KUKA KRL program: EPS_2_251455_MH14A_A_20251003045101.src

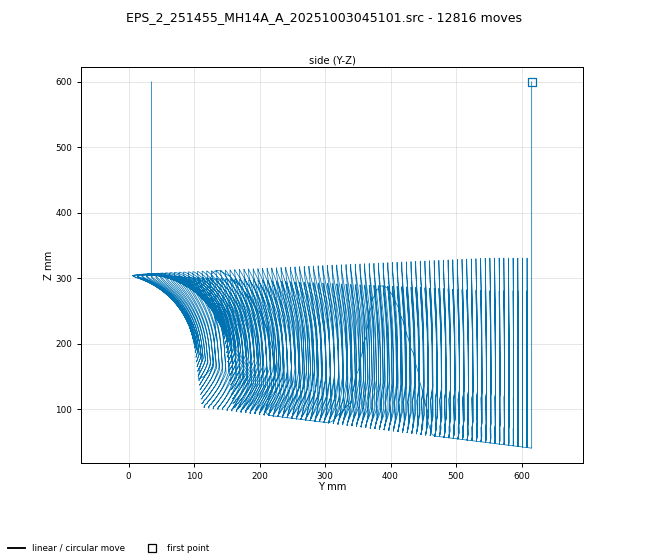
[picture p0: tool path of EPS_2_251455_MH14A_A_20251003045101.src, 12816 of 12818 moves have a stored position in this frame; points joined in program order, loops and branches not executed]
&ACCESS RVP
&REL 4
&COMMENT QRS 19112012
&PARAM EDITMASK = *
DEF PART()
EXT BAS (BAS_COMMAND :IN,REAL :IN )
INT I
BAS (#INITMOV,0 )

;KUKA QRS Post kuka4.cps  Date:22-06-2017 !

File_ID=2870

QRS_PRE_INIT()

;Init var - Until changes are made in qrs_pre_init
Outlet_Square_prg=0
Inlet_1_Square_prg=0
Inlet_2_Square_prg=0
Inlet_3_Square_prg=0
Inlet_4_Square_prg=0
Inlet_5_Square_prg=0

Outlet_1={X 0.000, Y 551.740, Z 230.500, B 0.000, E1 0.000 }
Inlet_1={X 0.000, Y 555.300, Z 180.500, B 0.000, E1 187.000 }
Outlet_1_type=201
Inlet_1_type=201
;QRS#1=Sidecore dimensions
;QRS#2=200-8" PVC SDR 35
;QRS#3=200-8" PVC SDR 35
;QRS#4=
;QRS#5=
;QRS#6=
;QRS#7=
;QRS#8=
;QRS#9=12-08 PSX
;QRS#10=12-08 PSX
;QRS#11=
;QRS#12=
;QRS#13=
;QRS#14=
;QRS#15=
;QRS#16=1220x127x610 2'
;QRS#17=EPS Height
;QRS#18=331
;QRS#19=*
;QRS#20= UPDATED VERSION 22-06-2017
;QRS#21=*
Outlet_Square=0100
Inlet_1_Square=0100
Inlet_2_Square=0
Inlet_3_Square=0
Inlet_4_Square=0
Inlet_5_Square=0
Mill_Square=1
Outlet_Square_Prg=204
Inlet_1_Square_prg=204

QRS_INIT()

$ADVANCE=5

; T1
PTP {E1 173.635,E2 173.635}
PTP {X 0,Y 615.458,A -85,B 0,C 180,E1 173.635,E2 173.635,E3 0,E4 0,E5 0,E6 0}
QRS_SPEED_INIT()
LIN {X 0,Y 615.458,Z 600,A -85,B 0,C 180,E1 173.635,E2 173.635,E3 0,E4 0,E5 0,E6 0} C_VEL
LIN {X 0,Y 615.458,Z 50.874,A -85,B 0,C 180,E1 173.635,E2 173.635} C_VEL
LIN {X 0,Y 615.458,Z 42.693,A -85,B 0,C 180,E1 173.635,E2 173.635} C_VEL
LIN {X 0,Y 615.454,Z 40.693,A -85,B 0,C 180,E1 173.449,E2 173.449} C_VEL
LIN {X 0,Y 615.495,Z 40.685,A -85,B 0,C 180,E1 170.801,E2 170.801} C_VEL
LIN {X 0,Y 615.481,Z 40.699,A -85,B 0,C 180,E1 168.139,E2 168.139} C_VEL
LIN {X 0,Y 615.455,Z 40.691,A -85,B 0,C 180,E1 165.45,E2 165.45} C_VEL
LIN {X 0,Y 615.493,Z 40.692,A -85,B 0,C 180,E1 162.729,E2 162.729} C_VEL
LIN {X 0,Y 615.454,Z 40.694,A -85,B 0,C 180,E1 159.966,E2 159.966} C_VEL
LIN {X 0,Y 615.455,Z 40.69,A -85,B 0,C 180,E1 157.661,E2 157.661} C_VEL
LIN {X 0,Y 615.495,Z 40.691,A -85,B 0,C 180,E1 155.008,E2 155.008} C_VEL
LIN {X 0,Y 615.45,Z 40.693,A -85,B 0,C 180,E1 152.083,E2 152.083} C_VEL
LIN {X 0,Y 615.452,Z 40.691,A -85,B 0,C 180,E1 149.838,E2 149.838} C_VEL
LIN {X 0,Y 615.478,Z 40.688,A -85,B 0,C 180,E1 147.542,E2 147.542} C_VEL
LIN {X 0,Y 615.495,Z 40.695,A -85,B 0,C 180,E1 145.185,E2 145.185} C_VEL
LIN {X 0,Y 615.465,Z 40.697,A -85,B 0,C 180,E1 142.756,E2 142.756} C_VEL
LIN {X 0,Y 615.448,Z 40.692,A -85,B 0,C 180,E1 140.246,E2 140.246} C_VEL
LIN {X 0,Y 615.499,Z 40.688,A -85,B 0,C 180,E1 137.647,E2 137.647} C_VEL
LIN {X 0,Y 615.458,Z 40.697,A -85,B 0,C 180,E1 134.928,E2 134.928} C_VEL
LIN {X 0,Y 615.451,Z 40.691,A -85,B 0,C 180,E1 132.356,E2 132.356} C_VEL
LIN {X 0,Y 615.495,Z 40.693,A -85,B 0,C 180,E1 129.749,E2 129.749} C_VEL
LIN {X 0,Y 615.445,Z 40.695,A -85,B 0,C 180,E1 126.931,E2 126.931} C_VEL
LIN {X 0,Y 615.444,Z 40.693,A -85,B 0,C 180,E1 124.694,E2 124.694} C_VEL
LIN {X 0,Y 615.472,Z 40.69,A -85,B 0,C 180,E1 122.328,E2 122.328} C_VEL
LIN {X 0,Y 615.455,Z 40.697,A -85,B 0,C 180,E1 119.408,E2 119.408} C_VEL
LIN {X 0,Y 615.439,Z 40.695,A -85,B 0,C 180,E1 117.035,E2 117.035} C_VEL
LIN {X 0,Y 615.491,Z 40.692,A -85,B 0,C 180,E1 114.272,E2 114.272} C_VEL
LIN {X 0,Y 615.497,Z 40.698,A -85,B 0,C 180,E1 112.136,E2 112.136} C_VEL
LIN {X 0,Y 615.487,Z 40.7,A -85,B 0,C 180,E1 110.033,E2 110.033} C_VEL
LIN {X 0,Y 615.47,Z 40.699,A -85,B 0,C 180,E1 107.957,E2 107.957} C_VEL
LIN {X 0,Y 615.457,Z 40.699,A -85,B 0,C 180,E1 105.906,E2 105.906} C_VEL
LIN {X 0,Y 615.451,Z 40.698,A -85,B 0,C 180,E1 103.875,E2 103.875} C_VEL
LIN {X 0,Y 615.446,Z 40.697,A -85,B 0,C 180,E1 101.861,E2 101.861} C_VEL
LIN {X 0,Y 615.467,Z 40.868,A -85,B 0,C 180,E1 100.958,E2 100.958} C_VEL
LIN {X 0,Y 615.443,Z 56.59,A -85,B 0,C 180,E1 98.206,E2 98.206} C_VEL
LIN {X 0,Y 615.459,Z 70.383,A -85,B 0,C 180,E1 95.816,E2 95.816} C_VEL
LIN {X 0,Y 615.474,Z 176.897,A -85,B 0,C 180,E1 94.543,E2 94.543} C_VEL
LIN {X 0,Y 615.468,Z 189.97,A -85,B 0,C 180,E1 94.256,E2 94.256} C_VEL
LIN {X 0,Y 615.485,Z 202.502,A -85,B 0,C 180,E1 93.846,E2 93.846} C_VEL
LIN {X 0,Y 615.485,Z 213.691,A -85,B 0,C 180,E1 93.355,E2 93.355} C_VEL
LIN {X 0,Y 615.491,Z 225.253,A -85,B 0,C 180,E1 92.7,E2 92.7} C_VEL
LIN {X 0,Y 615.498,Z 236.649,A -85,B 0,C 180,E1 91.881,E2 91.881} C_VEL
LIN {X 0,Y 615.498,Z 244.983,A -85,B 0,C 180,E1 91.145,E2 91.145} C_VEL
LIN {X 0,Y 615.498,Z 254.024,A -85,B 0,C 180,E1 90.163,E2 90.163} C_VEL
LIN {X 0,Y 615.498,Z 261.318,A -85,B 0,C 180,E1 89.182,E2 89.182} C_VEL
LIN {X 0,Y 615.497,Z 268.049,A -85,B 0,C 180,E1 88.037,E2 88.037} C_VEL
LIN {X 0,Y 615.496,Z 272.502,A -85,B 0,C 180,E1 87.054,E2 87.054} C_VEL
LIN {X 0,Y 615.496,Z 275.893,A -85,B 0,C 180,E1 86.071,E2 86.071} C_VEL
LIN {X 0,Y 615.498,Z 277.586,A -85,B 0,C 180,E1 85.415,E2 85.415} C_VEL
LIN {X 0,Y 615.497,Z 279.772,A -85,B 0,C 180,E1 84.101,E2 84.101} C_VEL
LIN {X 0,Y 615.495,Z 280.285,A -85,B 0,C 180,E1 83.42,E2 83.42} C_VEL
LIN {X 0,Y 615.494,Z 280.049,A -85,B 0,C 180,E1 82.124,E2 82.124} C_VEL
LIN {X 0,Y 615.496,Z 279.365,A -85,B 0,C 180,E1 81.463,E2 81.463} C_VEL
LIN {X 0,Y 615.496,Z 278.251,A -85,B 0,C 180,E1 80.801,E2 80.801} C_VEL
LIN {X 0,Y 615.496,Z 276.7,A -85,B 0,C 180,E1 80.138,E2 80.138} C_VEL
LIN {X 0,Y 615.496,Z 273.454,A -85,B 0,C 180,E1 79.11,E2 79.11} C_VEL
LIN {X 0,Y 615.496,Z 269.345,A -85,B 0,C 180,E1 78.139,E2 78.139} C_VEL
LIN {X 0,Y 615.496,Z 262.875,A -85,B 0,C 180,E1 76.967,E2 76.967} C_VEL
LIN {X 0,Y 615.497,Z 255.382,A -85,B 0,C 180,E1 75.912,E2 75.912} C_VEL
LIN {X 0,Y 615.498,Z 246.759,A -85,B 0,C 180,E1 74.943,E2 74.943} C_VEL
LIN {X 0,Y 615.497,Z 237.478,A -85,B 0,C 180,E1 74.095,E2 74.095} C_VEL
LIN {X 0,Y 615.487,Z 227.053,A -85,B 0,C 180,E1 73.328,E2 73.328} C_VEL
LIN {X 0,Y 615.468,Z 215.403,A -85,B 0,C 180,E1 72.643,E2 72.643} C_VEL
LIN {X 0,Y 615.492,Z 203.097,A -85,B 0,C 180,E1 72.086,E2 72.086} C_VEL
LIN {X 0,Y 615.489,Z 190.885,A -85,B 0,C 180,E1 71.679,E2 71.679} C_VEL
LIN {X 0,Y 615.489,Z 177.332,A -85,B 0,C 180,E1 71.375,E2 71.375} C_VEL
LIN {X 0,Y 615.475,Z 70.399,A -85,B 0,C 180,E1 70.097,E2 70.097} C_VEL
LIN {X 0,Y 615.495,Z 54.86,A -85,B 0,C 180,E1 67.405,E2 67.405} C_VEL
LIN {X 0,Y 615.436,Z 40.698,A -85,B 0,C 180,E1 64.901,E2 64.901} C_VEL
LIN {X 0,Y 615.428,Z 40.698,A -85,B 0,C 180,E1 62.82,E2 62.82} C_VEL
LIN {X 0,Y 615.428,Z 40.697,A -85,B 0,C 180,E1 60.59,E2 60.59} C_VEL
LIN {X 0,Y 615.446,Z 40.696,A -85,B 0,C 180,E1 58.312,E2 58.312} C_VEL
LIN {X 0,Y 615.494,Z 40.696,A -85,B 0,C 180,E1 55.978,E2 55.978} C_VEL
LIN {X 0,Y 615.454,Z 40.699,A -85,B 0,C 180,E1 53.573,E2 53.573} C_VEL
LIN {X 0,Y 615.42,Z 40.699,A -85,B 0,C 180,E1 50.946,E2 50.946} C_VEL
LIN {X 0,Y 615.449,Z 40.698,A -85,B 0,C 180,E1 48.523,E2 48.523} C_VEL
LIN {X 0,Y 615.452,Z 40.7,A -85,B 0,C 180,E1 45.847,E2 45.847} C_VEL
LIN {X 0,Y 615.461,Z 40.7,A -85,B 0,C 180,E1 43.995,E2 43.995} C_VEL
LIN {X 0,Y 615.415,Z 40.7,A -85,B 0,C 180,E1 41.48,E2 41.48} C_VEL
LIN {X 0,Y 615.438,Z 40.7,A -85,B 0,C 180,E1 38.909,E2 38.909} C_VEL
LIN {X 0,Y 615.469,Z 40.704,A -85,B 0,C 180,E1 36.426,E2 36.426} C_VEL
LIN {X 0,Y 615.435,Z 40.699,A -85,B 0,C 180,E1 34.026,E2 34.026} C_VEL
LIN {X 0,Y 615.419,Z 40.699,A -85,B 0,C 180,E1 31.69,E2 31.69} C_VEL
LIN {X 0,Y 615.426,Z 40.7,A -85,B 0,C 180,E1 29.41,E2 29.41} C_VEL
LIN {X 0,Y 615.473,Z 40.7,A -85,B 0,C 180,E1 27.042,E2 27.042} C_VEL
LIN {X 0,Y 615.437,Z 40.697,A -85,B 0,C 180,E1 24.274,E2 24.274} C_VEL
LIN {X 0,Y 615.428,Z 40.697,A -85,B 0,C 180,E1 22.139,E2 22.139} C_VEL
LIN {X 0,Y 615.426,Z 40.697,A -85,B 0,C 180,E1 20.035,E2 20.035} C_VEL
LIN {X 0,Y 615.486,Z 40.701,A -85,B 0,C 180,E1 17.271,E2 17.271} C_VEL
LIN {X 0,Y 615.439,Z 40.695,A -85,B 0,C 180,E1 14.55,E2 14.55} C_VEL
LIN {X 0,Y 615.437,Z 40.695,A -85,B 0,C 180,E1 12.531,E2 12.531} C_VEL
LIN {X 0,Y 615.436,Z 40.695,A -85,B 0,C 180,E1 10.528,E2 10.528} C_VEL
LIN {X 0,Y 615.435,Z 40.695,A -85,B 0,C 180,E1 8.538,E2 8.538} C_VEL
LIN {X 0,Y 615.459,Z 40.7,A -85,B 0,C 180,E1 5.899,E2 5.899} C_VEL
LIN {X 0,Y 615.478,Z 40.692,A -85,B 0,C 180,E1 3.273,E2 3.273} C_VEL
LIN {X 0,Y 615.438,Z 40.695,A -85,B 0,C 180,E1 0.654,E2 0.654} C_VEL
LIN {X 0,Y 615.481,Z 40.699,A -85,B 0,C 180,E1 -1.963,E2 -1.963} C_VEL
LIN {X 0,Y 615.473,Z 40.69,A -85,B 0,C 180,E1 -4.585,E2 -4.585} C_VEL
LIN {X 0,Y 615.443,Z 40.695,A -85,B 0,C 180,E1 -7.216,E2 -7.216} C_VEL
LIN {X 0,Y 615.499,Z 40.699,A -85,B 0,C 180,E1 -9.862,E2 -9.862} C_VEL
LIN {X 0,Y 615.46,Z 40.69,A -85,B 0,C 180,E1 -12.531,E2 -12.531} C_VEL
LIN {X 0,Y 615.456,Z 40.691,A -85,B 0,C 180,E1 -14.55,E2 -14.55} C_VEL
LIN {X 0,Y 615.45,Z 40.692,A -85,B 0,C 180,E1 -16.588,E2 -16.588} C_VEL
LIN {X 0,Y 615.448,Z 40.693,A -85,B 0,C 180,E1 -18.647,E2 -18.647} C_VEL
LIN {X 0,Y 615.497,Z 40.7,A -85,B 0,C 180,E1 -21.432,E2 -21.432} C_VEL
LIN {X 0,Y 615.459,Z 40.69,A -85,B 0,C 180,E1 -24.273,E2 -24.273} C_VEL
LIN {X 0,Y 615.453,Z 40.692,A -85,B 0,C 180,E1 -26.446,E2 -26.446} C_VEL
LIN {X 0,Y 615.458,Z 40.695,A -85,B 0,C 180,E1 -28.66,E2 -28.66} C_VEL
LIN {X 0,Y 615.486,Z 40.703,A -85,B 0,C 180,E1 -31.085,E2 -31.085} C_VEL
LIN {X 0,Y 615.461,Z 40.689,A -85,B 0,C 180,E1 -34.024,E2 -34.024} C_VEL
LIN {X 0,Y 615.463,Z 40.695,A -85,B 0,C 180,E1 -36.427,E2 -36.427} C_VEL
LIN {X 0,Y 615.492,Z 40.693,A -85,B 0,C 180,E1 -39.062,E2 -39.062} C_VEL
LIN {X 0,Y 615.487,Z 40.684,A -85,B 0,C 180,E1 -41.474,E2 -41.474} C_VEL
LIN {X 0,Y 615.463,Z 40.695,A -85,B 0,C 180,E1 -44.152,E2 -44.152} C_VEL
LIN {X 0,Y 615.489,Z 40.689,A -85,B 0,C 180,E1 -46.953,E2 -46.953} C_VEL
LIN {X 0,Y 615.474,Z 40.686,A -85,B 0,C 180,E1 -49.392,E2 -49.392} C_VEL
LIN {X 0,Y 615.469,Z 40.696,A -85,B 0,C 180,E1 -51.99,E2 -51.99} C_VEL
LIN {X 0,Y 615.493,Z 40.697,A -85,B 0,C 180,E1 -54.384,E2 -54.384} C_VEL
LIN {X 0,Y 615.486,Z 40.687,A -85,B 0,C 180,E1 -56.763,E2 -56.763} C_VEL
LIN {X 0,Y 615.478,Z 40.685,A -85,B 0,C 180,E1 -59.079,E2 -59.079} C_VEL
LIN {X 0,Y 615.471,Z 40.693,A -85,B 0,C 180,E1 -61.553,E2 -61.553} C_VEL
LIN {X 0,Y 615.487,Z 40.687,A -85,B 0,C 180,E1 -64.432,E2 -64.432} C_VEL
LIN {X 0,Y 615.47,Z 40.821,A -85,B 0,C 180,E1 -67.066,E2 -67.066} C_VEL
LIN {X 0,Y 615.461,Z 60.773,A -85,B 0,C 180,E1 -69.706,E2 -69.706} C_VEL
LIN {X 0,Y 615.488,Z 82.668,A -85,B 0,C 180,E1 -72.558,E2 -72.558} C_VEL
LIN {X 0,Y 615.467,Z 103.89,A -85,B 0,C 180,E1 -75.281,E2 -75.281} C_VEL
LIN {X 0,Y 615.452,Z 118.299,A -85,B 0,C 180,E1 -77.113,E2 -77.113} C_VEL
LIN {X 0,Y 615.492,Z 226.816,A -85,B 0,C 180,E1 -78.411,E2 -78.411} C_VEL
LIN {X 0,Y 615.48,Z 239.337,A -85,B 0,C 180,E1 -78.681,E2 -78.681} C_VEL
LIN {X 0,Y 615.489,Z 252.607,A -85,B 0,C 180,E1 -79.113,E2 -79.113} C_VEL
LIN {X 0,Y 615.475,Z 264.475,A -85,B 0,C 180,E1 -79.639,E2 -79.639} C_VEL
LIN {X 0,Y 615.492,Z 275.991,A -85,B 0,C 180,E1 -80.304,E2 -80.304} C_VEL
LIN {X 0,Y 615.499,Z 286.338,A -85,B 0,C 180,E1 -81.05,E2 -81.05} C_VEL
LIN {X 0,Y 615.497,Z 294.809,A -85,B 0,C 180,E1 -81.794,E2 -81.794} C_VEL
LIN {X 0,Y 615.498,Z 302.604,A -85,B 0,C 180,E1 -82.619,E2 -82.619} C_VEL
LIN {X 0,Y 615.496,Z 310.201,A -85,B 0,C 180,E1 -83.608,E2 -83.608} C_VEL
LIN {X 0,Y 615.498,Z 317.203,A -85,B 0,C 180,E1 -84.759,E2 -84.759} C_VEL
LIN {X 0,Y 615.493,Z 321.85,A -85,B 0,C 180,E1 -85.743,E2 -85.743} C_VEL
LIN {X 0,Y 615.494,Z 325.398,A -85,B 0,C 180,E1 -86.727,E2 -86.727} C_VEL
LIN {X 0,Y 615.497,Z 327.232,A -85,B 0,C 180,E1 -87.382,E2 -87.382} C_VEL
LIN {X 0,Y 615.5,Z 328.607,A -85,B 0,C 180,E1 -88.037,E2 -88.037} C_VEL
LIN {X 0,Y 615.496,Z 330.173,A -85,B 0,C 180,E1 -89.346,E2 -89.346} C_VEL
LIN {X 0,Y 615.494,Z 330.389,A -85,B 0,C 180,E1 -90,E2 -90} C_VEL
LIN {X 0,Y 615.495,Z 329.58,A -85,B 0,C 180,E1 -91.308,E2 -91.308} C_VEL
LIN {X 0,Y 615.5,Z 328.608,A -85,B 0,C 180,E1 -91.963,E2 -91.963} C_VEL
LIN {X 0,Y 615.497,Z 327.233,A -85,B 0,C 180,E1 -92.618,E2 -92.618} C_VEL
LIN {X 0,Y 615.496,Z 324.35,A -85,B 0,C 180,E1 -93.6,E2 -93.6} C_VEL
LIN {X 0,Y 615.498,Z 320.442,A -85,B 0,C 180,E1 -94.584,E2 -94.584} C_VEL
LIN {X 0,Y 615.499,Z 315.406,A -85,B 0,C 180,E1 -95.569,E2 -95.569} C_VEL
LIN {X 0,Y 615.497,Z 308.869,A -85,B 0,C 180,E1 -96.583,E2 -96.583} C_VEL
LIN {X 0,Y 615.497,Z 301.135,A -85,B 0,C 180,E1 -97.545,E2 -97.545} C_VEL
LIN {X 0,Y 615.498,Z 293.047,A -85,B 0,C 180,E1 -98.371,E2 -98.371} C_VEL
LIN {X 0,Y 615.499,Z 283.17,A -85,B 0,C 180,E1 -99.198,E2 -99.198} C_VEL
LIN {X 0,Y 615.484,Z 271.985,A -85,B 0,C 180,E1 -99.945,E2 -99.945} C_VEL
LIN {X 0,Y 615.481,Z 261.027,A -85,B 0,C 180,E1 -100.527,E2 -100.527} C_VEL
LIN {X 0,Y 615.481,Z 248.487,A -85,B 0,C 180,E1 -101.04,E2 -101.04} C_VEL
LIN {X 0,Y 615.482,Z 236.074,A -85,B 0,C 180,E1 -101.401,E2 -101.401} C_VEL
LIN {X 0,Y 615.497,Z 222.476,A -85,B 0,C 180,E1 -101.652,E2 -101.652} C_VEL
LIN {X 0,Y 615.452,Z 118.302,A -85,B 0,C 180,E1 -102.887,E2 -102.887} C_VEL
LIN {X 0,Y 615.488,Z 95.935,A -85,B 0,C 180,E1 -105.735,E2 -105.735} C_VEL
LIN {X 0,Y 615.456,Z 75.012,A -85,B 0,C 180,E1 -108.435,E2 -108.435} C_VEL
LIN {X 0,Y 615.489,Z 54.783,A -85,B 0,C 180,E1 -111.081,E2 -111.081} C_VEL
LIN {X 0,Y 615.472,Z 40.688,A -85,B 0,C 180,E1 -112.978,E2 -112.978} C_VEL
LIN {X 0,Y 615.485,Z 40.691,A -85,B 0,C 180,E1 -115.716,E2 -115.716} C_VEL
LIN {X 0,Y 615.473,Z 40.693,A -85,B 0,C 180,E1 -118.447,E2 -118.447} C_VEL
LIN {X 0,Y 615.485,Z 40.684,A -85,B 0,C 180,E1 -121.085,E2 -121.085} C_VEL
LIN {X 0,Y 615.483,Z 40.698,A -85,B 0,C 180,E1 -124.022,E2 -124.022} C_VEL
LIN {X 0,Y 615.468,Z 40.69,A -85,B 0,C 180,E1 -126.426,E2 -126.426} C_VEL
LIN {X 0,Y 615.492,Z 40.685,A -85,B 0,C 180,E1 -129.062,E2 -129.062} C_VEL
LIN {X 0,Y 615.49,Z 40.697,A -85,B 0,C 180,E1 -131.473,E2 -131.473} C_VEL
LIN {X 0,Y 615.467,Z 40.691,A -85,B 0,C 180,E1 -134.151,E2 -134.151} C_VEL
LIN {X 0,Y 615.487,Z 40.688,A -85,B 0,C 180,E1 -136.952,E2 -136.952} C_VEL
LIN {X 0,Y 615.486,Z 40.702,A -85,B 0,C 180,E1 -139.393,E2 -139.393} C_VEL
LIN {X 0,Y 615.465,Z 40.69,A -85,B 0,C 180,E1 -141.991,E2 -141.991} C_VEL
LIN {X 0,Y 615.489,Z 40.683,A -85,B 0,C 180,E1 -144.384,E2 -144.384} C_VEL
LIN {X 0,Y 615.489,Z 40.691,A -85,B 0,C 180,E1 -146.764,E2 -146.764} C_VEL
LIN {X 0,Y 615.49,Z 40.702,A -85,B 0,C 180,E1 -149.08,E2 -149.08} C_VEL
LIN {X 0,Y 615.464,Z 40.692,A -85,B 0,C 180,E1 -151.554,E2 -151.554} C_VEL
LIN {X 0,Y 615.496,Z 40.684,A -85,B 0,C 180,E1 -154.285,E2 -154.285} C_VEL
LIN {X 0,Y 615.471,Z 40.696,A -85,B 0,C 180,E1 -157.155,E2 -157.155} C_VEL
LIN {X 0,Y 615.483,Z 40.685,A -85,B 0,C 180,E1 -159.967,E2 -159.967} C_VEL
LIN {X 0,Y 615.49,Z 40.699,A -85,B 0,C 180,E1 -162.73,E2 -162.73} C_VEL
LIN {X 0,Y 615.464,Z 40.689,A -85,B 0,C 180,E1 -165.45,E2 -165.45} C_VEL
LIN {X 0,Y 615.491,Z 40.691,A -85,B 0,C 180,E1 -168.139,E2 -168.139} C_VEL
LIN {X 0,Y 615.465,Z 40.695,A -85,B 0,C 180,E1 -170.801,E2 -170.801} C_VEL
LIN {X 0,Y 615.476,Z 40.686,A -85,B 0,C 180,E1 -173.443,E2 -173.443} C_VEL
LIN {X 0,Y 615.492,Z 40.697,A -85,B 0,C 180,E1 -176.072,E2 -176.072} C_VEL
LIN {X 0,Y 615.457,Z 40.694,A -85,B 0,C 180,E1 -178.691,E2 -178.691} C_VEL
LIN {X 0,Y 615.483,Z 40.685,A -85,B 0,C 180,E1 -181.309,E2 -181.309} C_VEL
LIN {X 0,Y 615.488,Z 40.701,A -85,B 0,C 180,E1 -183.929,E2 -183.929} C_VEL
LIN {X 0,Y 615.454,Z 40.693,A -85,B 0,C 180,E1 -186.551,E2 -186.551} C_VEL
LIN {X 0,Y 614.802,Z 40.835,A -85,B 0,C 180,E1 -187.097,E2 -187.097} C_VEL
LIN {X 0,Y 611.99,Z 41.255,A -85,B 0,C 180,E1 -187.984,E2 -187.984} C_VEL
LIN {X 0,Y 609.6,Z 41.562,A -85,B 0,C 180,E1 -188.696,E2 -188.696} C_VEL
LIN {X 0,Y 608.559,Z 41.678,A -85,B 0,C 180,E1 -189.246,E2 -189.246} C_VEL
LIN {X 0,Y 608.467,Z 41.689,A -85,B 0,C 180,E1 -189.432,E2 -189.432} C_VEL
LIN {X 0,Y 608.452,Z 41.693,A -85,B 0,C 180,E1 -192,E2 -192} C_VEL
LIN {X 0,Y 608.429,Z 41.691,A -85,B 0,C 180,E1 -194.722,E2 -194.722} C_VEL
LIN {X 0,Y 608.45,Z 41.697,A -85,B 0,C 180,E1 -197.477,E2 -197.477} C_VEL
LIN {X 0,Y 608.437,Z 41.69,A -85,B 0,C 180,E1 -200.275,E2 -200.275} C_VEL
LIN {X 0,Y 608.429,Z 41.691,A -85,B 0,C 180,E1 -202.47,E2 -202.47} C_VEL
LIN {X 0,Y 608.446,Z 41.699,A -85,B 0,C 180,E1 -205.302,E2 -205.302} C_VEL
LIN {X 0,Y 608.437,Z 41.695,A -85,B 0,C 180,E1 -207.519,E2 -207.519} C_VEL
LIN {X 0,Y 608.418,Z 41.692,A -85,B 0,C 180,E1 -209.964,E2 -209.964} C_VEL
LIN {X 0,Y 608.455,Z 41.69,A -85,B 0,C 180,E1 -212.522,E2 -212.522} C_VEL
LIN {X 0,Y 608.427,Z 41.696,A -85,B 0,C 180,E1 -215.279,E2 -215.279} C_VEL
LIN {X 0,Y 608.446,Z 41.689,A -85,B 0,C 180,E1 -217.748,E2 -217.748} C_VEL
LIN {X 0,Y 608.443,Z 41.692,A -85,B 0,C 180,E1 -220.328,E2 -220.328} C_VEL
LIN {X 0,Y 608.437,Z 41.696,A -85,B 0,C 180,E1 -222.962,E2 -222.962} C_VEL
LIN {X 0,Y 608.431,Z 41.69,A -85,B 0,C 180,E1 -225.739,E2 -225.739} C_VEL
LIN {X 0,Y 608.451,Z 41.689,A -85,B 0,C 180,E1 -227.938,E2 -227.938} C_VEL
LIN {X 0,Y 608.43,Z 41.697,A -85,B 0,C 180,E1 -230.708,E2 -230.708} C_VEL
LIN {X 0,Y 608.416,Z 41.693,A -85,B 0,C 180,E1 -233.082,E2 -233.082} C_VEL
LIN {X 0,Y 608.446,Z 41.689,A -85,B 0,C 180,E1 -235.529,E2 -235.529} C_VEL
LIN {X 0,Y 608.458,Z 41.691,A -85,B 0,C 180,E1 -237.905,E2 -237.905} C_VEL
LIN {X 0,Y 608.482,Z 41.694,A -85,B 0,C 180,E1 -240.221,E2 -240.221} C_VEL
LIN {X 0,Y 608.421,Z 41.693,A -85,B 0,C 180,E1 -242.804,E2 -242.804} C_VEL
LIN {X 0,Y 608.44,Z 41.691,A -85,B 0,C 180,E1 -245.429,E2 -245.429} C_VEL
LIN {X 0,Y 608.448,Z 41.692,A -85,B 0,C 180,E1 -248.308,E2 -248.308} C_VEL
LIN {X 0,Y 608.425,Z 41.693,A -85,B 0,C 180,E1 -250.429,E2 -250.429} C_VEL
LIN {X 0,Y 608.436,Z 41.692,A -85,B 0,C 180,E1 -253.216,E2 -253.216} C_VEL
LIN {X 0,Y 608.435,Z 41.695,A -85,B 0,C 180,E1 -255.998,E2 -255.998} C_VEL
LIN {X 0,Y 608.437,Z 41.694,A -85,B 0,C 180,E1 -258,E2 -258} C_VEL
LIN {X 0,Y 608.468,Z 41.758,A -85,B 0,C 180,E1 -258.971,E2 -258.971} C_VEL
LIN {X 0,Y 608.433,Z 57.206,A -85,B 0,C 180,E1 -261.698,E2 -261.698} C_VEL
LIN {X 0,Y 608.433,Z 70.587,A -85,B 0,C 180,E1 -264.033,E2 -264.033} C_VEL
LIN {X 0,Y 608.55,Z 153.667,A -85,B 0,C 180,E1 -265.031,E2 -265.031} C_VEL
LIN {X 0,Y 608.52,Z 178.093,A -85,B 0,C 180,E1 -265.342,E2 -265.342} C_VEL
LIN {X 0,Y 608.528,Z 191.538,A -85,B 0,C 180,E1 -265.653,E2 -265.653} C_VEL
LIN {X 0,Y 608.513,Z 203.71,A -85,B 0,C 180,E1 -266.068,E2 -266.068} C_VEL
LIN {X 0,Y 608.493,Z 215.437,A -85,B 0,C 180,E1 -266.607,E2 -266.607} C_VEL
LIN {X 0,Y 608.495,Z 226.702,A -85,B 0,C 180,E1 -267.269,E2 -267.269} C_VEL
LIN {X 0,Y 608.472,Z 236.896,A -85,B 0,C 180,E1 -268.014,E2 -268.014} C_VEL
LIN {X 0,Y 608.479,Z 246.116,A -85,B 0,C 180,E1 -268.842,E2 -268.842} C_VEL
LIN {X 0,Y 608.469,Z 255.057,A -85,B 0,C 180,E1 -269.835,E2 -269.835} C_VEL
LIN {X 0,Y 608.448,Z 262.293,A -85,B 0,C 180,E1 -270.827,E2 -270.827} C_VEL
LIN {X 0,Y 608.443,Z 268.932,A -85,B 0,C 180,E1 -271.986,E2 -271.986} C_VEL
LIN {X 0,Y 608.451,Z 273.336,A -85,B 0,C 180,E1 -272.98,E2 -272.98} C_VEL
LIN {X 0,Y 608.433,Z 276.683,A -85,B 0,C 180,E1 -273.974,E2 -273.974} C_VEL
LIN {X 0,Y 608.431,Z 278.346,A -85,B 0,C 180,E1 -274.638,E2 -274.638} C_VEL
LIN {X 0,Y 608.433,Z 280.473,A -85,B 0,C 180,E1 -275.967,E2 -275.967} C_VEL
LIN {X 0,Y 608.43,Z 280.91,A -85,B 0,C 180,E1 -276.633,E2 -276.633} C_VEL
LIN {X 0,Y 608.419,Z 280.6,A -85,B 0,C 180,E1 -277.968,E2 -277.968} C_VEL
LIN {X 0,Y 608.422,Z 279.854,A -85,B 0,C 180,E1 -278.637,E2 -278.637} C_VEL
LIN {X 0,Y 608.421,Z 278.659,A -85,B 0,C 180,E1 -279.307,E2 -279.307} C_VEL
LIN {X 0,Y 608.433,Z 276.089,A -85,B 0,C 180,E1 -280.314,E2 -280.314} C_VEL
LIN {X 0,Y 608.43,Z 272.482,A -85,B 0,C 180,E1 -281.325,E2 -281.325} C_VEL
LIN {X 0,Y 608.459,Z 267.726,A -85,B 0,C 180,E1 -282.339,E2 -282.339} C_VEL
LIN {X 0,Y 608.459,Z 260.513,A -85,B 0,C 180,E1 -283.527,E2 -283.527} C_VEL
LIN {X 0,Y 608.459,Z 252.619,A -85,B 0,C 180,E1 -284.55,E2 -284.55} C_VEL
LIN {X 0,Y 608.467,Z 244.475,A -85,B 0,C 180,E1 -285.406,E2 -285.406} C_VEL
LIN {X 0,Y 608.49,Z 234.985,A -85,B 0,C 180,E1 -286.226,E2 -286.226} C_VEL
LIN {X 0,Y 608.483,Z 224.636,A -85,B 0,C 180,E1 -286.956,E2 -286.956} C_VEL
LIN {X 0,Y 608.48,Z 213.912,A -85,B 0,C 180,E1 -287.563,E2 -287.563} C_VEL
LIN {X 0,Y 608.512,Z 202.09,A -85,B 0,C 180,E1 -288.083,E2 -288.083} C_VEL
LIN {X 0,Y 608.538,Z 189.368,A -85,B 0,C 180,E1 -288.497,E2 -288.497} C_VEL
LIN {X 0,Y 608.559,Z 176.227,A -85,B 0,C 180,E1 -288.78,E2 -288.78} C_VEL
LIN {X 0,Y 608.44,Z 70.598,A -85,B 0,C 180,E1 -290.055,E2 -290.055} C_VEL
LIN {X 0,Y 608.469,Z 55.08,A -85,B 0,C 180,E1 -292.764,E2 -292.764} C_VEL
LIN {X 0,Y 608.425,Z 41.693,A -85,B 0,C 180,E1 -295.142,E2 -295.142} C_VEL
LIN {X 0,Y 608.416,Z 41.693,A -85,B 0,C 180,E1 -297.52,E2 -297.52} C_VEL
LIN {X 0,Y 608.451,Z 41.693,A -85,B 0,C 180,E1 -299.968,E2 -299.968} C_VEL
LIN {X 0,Y 608.422,Z 41.693,A -85,B 0,C 180,E1 -302.882,E2 -302.882} C_VEL
LIN {X 0,Y 608.405,Z 41.694,A -85,B 0,C 180,E1 -305.281,E2 -305.281} C_VEL
LIN {X 0,Y 608.427,Z 41.698,A -85,B 0,C 180,E1 -308.235,E2 -308.235} C_VEL
LIN {X 0,Y 608.397,Z 41.695,A -85,B 0,C 180,E1 -311.182,E2 -311.182} C_VEL
LIN {X 0,Y 608.452,Z 41.697,A -85,B 0,C 180,E1 -313.871,E2 -313.871} C_VEL
LIN {X 0,Y 608.412,Z 41.693,A -85,B 0,C 180,E1 -316.697,E2 -316.697} C_VEL
LIN {X 0,Y 608.387,Z 41.696,A -85,B 0,C 180,E1 -318.817,E2 -318.817} C_VEL
LIN {X 0,Y 608.399,Z 41.702,A -85,B 0,C 180,E1 -321.406,E2 -321.406} C_VEL
LIN {X 0,Y 608.429,Z 41.693,A -85,B 0,C 180,E1 -323.957,E2 -323.957} C_VEL
LIN {X 0,Y 608.414,Z 41.693,A -85,B 0,C 180,E1 -326.326,E2 -326.326} C_VEL
LIN {X 0,Y 608.432,Z 41.692,A -85,B 0,C 180,E1 -328.735,E2 -328.735} C_VEL
LIN {X 0,Y 608.414,Z 41.695,A -85,B 0,C 180,E1 -331.731,E2 -331.731} C_VEL
LIN {X 0,Y 608.403,Z 41.694,A -85,B 0,C 180,E1 -334.293,E2 -334.293} C_VEL
LIN {X 0,Y 608.43,Z 41.699,A -85,B 0,C 180,E1 -336.875,E2 -336.875} C_VEL
LIN {X 0,Y 608.418,Z 41.692,A -85,B 0,C 180,E1 -339.724,E2 -339.724} C_VEL
LIN {X 0,Y 608.401,Z 41.694,A -85,B 0,C 180,E1 -341.826,E2 -341.826} C_VEL
LIN {X 0,Y 608.46,Z 41.695,A -85,B 0,C 180,E1 -344.594,E2 -344.594} C_VEL
LIN {X 0,Y 608.418,Z 41.693,A -85,B 0,C 180,E1 -347.322,E2 -347.322} C_VEL
LIN {X 0,Y 608.425,Z 41.692,A -85,B 0,C 180,E1 -349.349,E2 -349.349} C_VEL
LIN {X 0,Y 608.419,Z 41.692,A -85,B 0,C 180,E1 -351.363,E2 -351.363} C_VEL
LIN {X 0,Y 608.432,Z 41.695,A -85,B 0,C 180,E1 -354.033,E2 -354.033} C_VEL
LIN {X 0,Y 608.471,Z 41.689,A -85,B 0,C 180,E1 -356.689,E2 -356.689} C_VEL
LIN {X 0,Y 608.417,Z 41.692,A -85,B 0,C 180,E1 -359.338,E2 -359.338} C_VEL
LIN {X 0,Y 608.45,Z 41.696,A -85,B 0,C 180,E1 -361.986,E2 -361.986} C_VEL
LIN {X 0,Y 608.439,Z 41.691,A -85,B 0,C 180,E1 -364.638,E2 -364.638} C_VEL
LIN {X 0,Y 608.422,Z 41.693,A -85,B 0,C 180,E1 -367.3,E2 -367.3} C_VEL
LIN {X 0,Y 608.463,Z 41.694,A -85,B 0,C 180,E1 -369.977,E2 -369.977} C_VEL
LIN {X 0,Y 608.45,Z 41.688,A -85,B 0,C 180,E1 -372.677,E2 -372.677} C_VEL
LIN {X 0,Y 608.456,Z 41.694,A -85,B 0,C 180,E1 -375.406,E2 -375.406} C_VEL
LIN {X 0,Y 608.442,Z 41.69,A -85,B 0,C 180,E1 -378.172,E2 -378.172} C_VEL
LIN {X 0,Y 608.442,Z 41.692,A -85,B 0,C 180,E1 -380.982,E2 -380.982} C_VEL
LIN {X 0,Y 608.464,Z 41.689,A -85,B 0,C 180,E1 -383.845,E2 -383.845} C_VEL
LIN {X 0,Y 608.437,Z 41.69,A -85,B 0,C 180,E1 -386.036,E2 -386.036} C_VEL
LIN {X 0,Y 608.448,Z 41.69,A -85,B 0,C 180,E1 -388.615,E2 -388.615} C_VEL
LIN {X 0,Y 608.449,Z 41.694,A -85,B 0,C 180,E1 -391.318,E2 -391.318} C_VEL
LIN {X 0,Y 608.476,Z 41.685,A -85,B 0,C 180,E1 -393.735,E2 -393.735} C_VEL
LIN {X 0,Y 608.441,Z 41.689,A -85,B 0,C 180,E1 -396.093,E2 -396.093} C_VEL
LIN {X 0,Y 608.435,Z 41.696,A -85,B 0,C 180,E1 -398.591,E2 -398.591} C_VEL
LIN {X 0,Y 608.465,Z 41.688,A -85,B 0,C 180,E1 -401.342,E2 -401.342} C_VEL
LIN {X 0,Y 608.452,Z 41.689,A -85,B 0,C 180,E1 -403.871,E2 -403.871} C_VEL
LIN {X 0,Y 608.477,Z 41.692,A -85,B 0,C 180,E1 -406.691,E2 -406.691} C_VEL
LIN {X 0,Y 608.46,Z 41.691,A -85,B 0,C 180,E1 -408.823,E2 -408.823} C_VEL
LIN {X 0,Y 608.44,Z 41.689,A -85,B 0,C 180,E1 -411.409,E2 -411.409} C_VEL
LIN {X 0,Y 608.447,Z 41.694,A -85,B 0,C 180,E1 -413.955,E2 -413.955} C_VEL
LIN {X 0,Y 608.453,Z 41.696,A -85,B 0,C 180,E1 -416.328,E2 -416.328} C_VEL
LIN {X 0,Y 608.45,Z 41.69,A -85,B 0,C 180,E1 -418.732,E2 -418.732} C_VEL
LIN {X 0,Y 608.46,Z 41.689,A -85,B 0,C 180,E1 -421.383,E2 -421.383} C_VEL
LIN {X 0,Y 608.441,Z 41.699,A -85,B 0,C 180,E1 -423.964,E2 -423.964} C_VEL
LIN {X 0,Y 608.471,Z 41.692,A -85,B 0,C 180,E1 -426.155,E2 -426.155} C_VEL
LIN {X 0,Y 608.474,Z 41.818,A -85,B 0,C 180,E1 -426.922,E2 -426.922} C_VEL
LIN {X 0,Y 608.585,Z 57.441,A -85,B 0,C 180,E1 -429.023,E2 -429.023} C_VEL
LIN {X 0,Y 608.522,Z 78.715,A -85,B 0,C 180,E1 -431.83,E2 -431.83} C_VEL
LIN {X 0,Y 608.496,Z 99.988,A -85,B 0,C 180,E1 -434.594,E2 -434.594} C_VEL
LIN {X 0,Y 608.45,Z 118.52,A -85,B 0,C 180,E1 -436.972,E2 -436.972} C_VEL
LIN {X 0,Y 608.549,Z 226.934,A -85,B 0,C 180,E1 -438.276,E2 -438.276} C_VEL
LIN {X 0,Y 608.515,Z 240.208,A -85,B 0,C 180,E1 -438.571,E2 -438.571} C_VEL
LIN {X 0,Y 608.515,Z 252.621,A -85,B 0,C 180,E1 -438.982,E2 -438.982} C_VEL
LIN {X 0,Y 608.498,Z 264.63,A -85,B 0,C 180,E1 -439.519,E2 -439.519} C_VEL
LIN {X 0,Y 608.48,Z 276.194,A -85,B 0,C 180,E1 -440.191,E2 -440.191} C_VEL
LIN {X 0,Y 608.485,Z 286.591,A -85,B 0,C 180,E1 -440.946,E2 -440.946} C_VEL
LIN {X 0,Y 608.475,Z 295.109,A -85,B 0,C 180,E1 -441.699,E2 -441.699} C_VEL
LIN {X 0,Y 608.471,Z 302.958,A -85,B 0,C 180,E1 -442.534,E2 -442.534} C_VEL
LIN {X 0,Y 608.461,Z 310.286,A -85,B 0,C 180,E1 -443.484,E2 -443.484} C_VEL
LIN {X 0,Y 608.451,Z 315.865,A -85,B 0,C 180,E1 -444.365,E2 -444.365} C_VEL
LIN {X 0,Y 608.432,Z 320.949,A -85,B 0,C 180,E1 -445.362,E2 -445.362} C_VEL
LIN {X 0,Y 608.449,Z 324.895,A -85,B 0,C 180,E1 -446.357,E2 -446.357} C_VEL
LIN {X 0,Y 608.425,Z 327.809,A -85,B 0,C 180,E1 -447.352,E2 -447.352} C_VEL
LIN {X 0,Y 608.444,Z 329.201,A -85,B 0,C 180,E1 -448.014,E2 -448.014} C_VEL
LIN {X 0,Y 608.439,Z 330.783,A -85,B 0,C 180,E1 -449.338,E2 -449.338} C_VEL
LIN {X 0,Y 608.434,Z 331,A -85,B 0,C 180,E1 -450,E2 -450} C_VEL
LIN {X 0,Y 608.448,Z 330.184,A -85,B 0,C 180,E1 -451.324,E2 -451.324} C_VEL
LIN {X 0,Y 608.445,Z 329.202,A -85,B 0,C 180,E1 -451.986,E2 -451.986} C_VEL
LIN {X 0,Y 608.425,Z 327.81,A -85,B 0,C 180,E1 -452.648,E2 -452.648} C_VEL
LIN {X 0,Y 608.449,Z 324.897,A -85,B 0,C 180,E1 -453.642,E2 -453.642} C_VEL
LIN {X 0,Y 608.432,Z 320.951,A -85,B 0,C 180,E1 -454.638,E2 -454.638} C_VEL
LIN {X 0,Y 608.438,Z 314.878,A -85,B 0,C 180,E1 -455.801,E2 -455.801} C_VEL
LIN {X 0,Y 608.462,Z 308.236,A -85,B 0,C 180,E1 -456.799,E2 -456.799} C_VEL
LIN {X 0,Y 608.456,Z 299.991,A -85,B 0,C 180,E1 -457.8,E2 -457.8} C_VEL
LIN {X 0,Y 608.472,Z 291.538,A -85,B 0,C 180,E1 -458.636,E2 -458.636} C_VEL
LIN {X 0,Y 608.479,Z 281.094,A -85,B 0,C 180,E1 -459.473,E2 -459.473} C_VEL
LIN {X 0,Y 608.486,Z 270.759,A -85,B 0,C 180,E1 -460.145,E2 -460.145} C_VEL
LIN {X 0,Y 608.519,Z 259.267,A -85,B 0,C 180,E1 -460.74,E2 -460.74} C_VEL
LIN {X 0,Y 608.529,Z 246.894,A -85,B 0,C 180,E1 -461.225,E2 -461.225} C_VEL
LIN {X 0,Y 608.547,Z 233.446,A -85,B 0,C 180,E1 -461.597,E2 -461.597} C_VEL
LIN {X 0,Y 608.554,Z 221.098,A -85,B 0,C 180,E1 -461.808,E2 -461.808} C_VEL
LIN {X 0,Y 608.438,Z 118.44,A -85,B 0,C 180,E1 -463.038,E2 -463.038} C_VEL
LIN {X 0,Y 608.506,Z 96.003,A -85,B 0,C 180,E1 -465.92,E2 -465.92} C_VEL
LIN {X 0,Y 608.5,Z 76.262,A -85,B 0,C 180,E1 -468.492,E2 -468.492} C_VEL
LIN {X 0,Y 608.567,Z 56.114,A -85,B 0,C 180,E1 -471.155,E2 -471.155} C_VEL
LIN {X 0,Y 608.465,Z 41.688,A -85,B 0,C 180,E1 -473.101,E2 -473.101} C_VEL
LIN {X 0,Y 608.471,Z 41.689,A -85,B 0,C 180,E1 -475.72,E2 -475.72} C_VEL
LIN {X 0,Y 608.443,Z 41.695,A -85,B 0,C 180,E1 -478.267,E2 -478.267} C_VEL
LIN {X 0,Y 608.465,Z 41.688,A -85,B 0,C 180,E1 -480.545,E2 -480.545} C_VEL
LIN {X 0,Y 608.451,Z 41.688,A -85,B 0,C 180,E1 -482.88,E2 -482.88} C_VEL
LIN {X 0,Y 608.443,Z 41.691,A -85,B 0,C 180,E1 -485.277,E2 -485.277} C_VEL
LIN {X 0,Y 608.464,Z 41.697,A -85,B 0,C 180,E1 -487.746,E2 -487.746} C_VEL
LIN {X 0,Y 608.437,Z 41.691,A -85,B 0,C 180,E1 -490.327,E2 -490.327} C_VEL
LIN {X 0,Y 608.452,Z 41.689,A -85,B 0,C 180,E1 -492.96,E2 -492.96} C_VEL
LIN {X 0,Y 608.441,Z 41.695,A -85,B 0,C 180,E1 -495.737,E2 -495.737} C_VEL
LIN {X 0,Y 608.448,Z 41.691,A -85,B 0,C 180,E1 -497.937,E2 -497.937} C_VEL
LIN {X 0,Y 608.444,Z 41.69,A -85,B 0,C 180,E1 -500.705,E2 -500.705} C_VEL
LIN {X 0,Y 608.454,Z 41.695,A -85,B 0,C 180,E1 -503.085,E2 -503.085} C_VEL
LIN {X 0,Y 608.466,Z 41.691,A -85,B 0,C 180,E1 -505.53,E2 -505.53} C_VEL
LIN {X 0,Y 608.454,Z 41.688,A -85,B 0,C 180,E1 -507.905,E2 -507.905} C_VEL
LIN {X 0,Y 608.47,Z 41.686,A -85,B 0,C 180,E1 -510.221,E2 -510.221} C_VEL
LIN {X 0,Y 608.444,Z 41.694,A -85,B 0,C 180,E1 -513.225,E2 -513.225} C_VEL
LIN {X 0,Y 608.469,Z 41.686,A -85,B 0,C 180,E1 -515.849,E2 -515.849} C_VEL
LIN {X 0,Y 608.468,Z 41.689,A -85,B 0,C 180,E1 -518.308,E2 -518.308} C_VEL
LIN {X 0,Y 608.456,Z 41.689,A -85,B 0,C 180,E1 -521.288,E2 -521.288} C_VEL
LIN {X 0,Y 608.457,Z 41.688,A -85,B 0,C 180,E1 -523.906,E2 -523.906} C_VEL
LIN {X 0,Y 608.456,Z 41.695,A -85,B 0,C 180,E1 -526.643,E2 -526.643} C_VEL
LIN {X 0,Y 608.446,Z 41.689,A -85,B 0,C 180,E1 -529.35,E2 -529.35} C_VEL
LIN {X 0,Y 608.479,Z 41.689,A -85,B 0,C 180,E1 -532.033,E2 -532.033} C_VEL
LIN {X 0,Y 608.445,Z 41.692,A -85,B 0,C 180,E1 -534.698,E2 -534.698} C_VEL
LIN {X 0,Y 608.471,Z 41.686,A -85,B 0,C 180,E1 -537.352,E2 -537.352} C_VEL
LIN {X 0,Y 608.481,Z 41.693,A -85,B 0,C 180,E1 -540,E2 -540} C_VEL
LIN {X 0,Y 608.451,Z 41.689,A -85,B 0,C 180,E1 -542.648,E2 -542.648} C_VEL
LIN {X 0,Y 608.468,Z 41.687,A -85,B 0,C 180,E1 -545.302,E2 -545.302} C_VEL
LIN {X 0,Y 608.473,Z 41.693,A -85,B 0,C 180,E1 -547.967,E2 -547.967} C_VEL
LIN {X 0,Y 608.467,Z 41.689,A -85,B 0,C 180,E1 -549.432,E2 -549.432} C_VEL
LIN {X 0,Y 607.779,Z 41.779,A -85,B 0,C 180,E1 -549.985,E2 -549.985} C_VEL
LIN {X 0,Y 604.921,Z 42.134,A -85,B 0,C 180,E1 -550.881,E2 -550.881} C_VEL
LIN {X 0,Y 602.517,Z 42.435,A -85,B 0,C 180,E1 -551.603,E2 -551.603} C_VEL
LIN {X 0,Y 601.484,Z 42.559,A -85,B 0,C 180,E1 -552.159,E2 -552.159} C_VEL
LIN {X 0,Y 601.398,Z 42.568,A -85,B 0,C 180,E1 -552.348,E2 -552.348} C_VEL
LIN {X 0,Y 601.401,Z 42.567,A -85,B 0,C 180,E1 -554.898,E2 -554.898} C_VEL
LIN {X 0,Y 601.41,Z 42.567,A -85,B 0,C 180,E1 -556.987,E2 -556.987} C_VEL
LIN {X 0,Y 601.395,Z 42.571,A -85,B 0,C 180,E1 -559.81,E2 -559.81} C_VEL
LIN {X 0,Y 601.403,Z 42.567,A -85,B 0,C 180,E1 -562.684,E2 -562.684} C_VEL
LIN {X 0,Y 601.419,Z 42.569,A -85,B 0,C 180,E1 -565.618,E2 -565.618} C_VEL
LIN {X 0,Y 601.389,Z 42.569,A -85,B 0,C 180,E1 -567.869,E2 -567.869} C_VEL
LIN {X 0,Y 601.399,Z 42.566,A -85,B 0,C 180,E1 -570.166,E2 -570.166} C_VEL
LIN {X 0,Y 601.416,Z 42.569,A -85,B 0,C 180,E1 -572.715,E2 -572.715} C_VEL
LIN {X 0,Y 601.393,Z 42.575,A -85,B 0,C 180,E1 -575.112,E2 -575.112} C_VEL
LIN {X 0,Y 601.43,Z 42.565,A -85,B 0,C 180,E1 -577.42,E2 -577.42} C_VEL
LIN {X 0,Y 601.397,Z 42.567,A -85,B 0,C 180,E1 -579.997,E2 -579.997} C_VEL
LIN {X 0,Y 601.41,Z 42.574,A -85,B 0,C 180,E1 -582.671,E2 -582.671} C_VEL
LIN {X 0,Y 601.401,Z 42.566,A -85,B 0,C 180,E1 -585.48,E2 -585.48} C_VEL
LIN {X 0,Y 601.42,Z 42.571,A -85,B 0,C 180,E1 -588.408,E2 -588.408} C_VEL
LIN {X 0,Y 601.392,Z 42.571,A -85,B 0,C 180,E1 -590.872,E2 -590.872} C_VEL
LIN {X 0,Y 601.393,Z 42.568,A -85,B 0,C 180,E1 -593.741,E2 -593.741} C_VEL
LIN {X 0,Y 601.41,Z 42.569,A -85,B 0,C 180,E1 -596.686,E2 -596.686} C_VEL
LIN {X 0,Y 601.403,Z 42.566,A -85,B 0,C 180,E1 -599.057,E2 -599.057} C_VEL
LIN {X 0,Y 601.41,Z 42.565,A -85,B 0,C 180,E1 -601.372,E2 -601.372} C_VEL
LIN {X 0,Y 601.399,Z 42.571,A -85,B 0,C 180,E1 -604.381,E2 -604.381} C_VEL
LIN {X 0,Y 601.38,Z 42.57,A -85,B 0,C 180,E1 -606.588,E2 -606.588} C_VEL
LIN {X 0,Y 601.428,Z 42.566,A -85,B 0,C 180,E1 -609.478,E2 -609.478} C_VEL
LIN {X 0,Y 601.373,Z 42.572,A -85,B 0,C 180,E1 -612.311,E2 -612.311} C_VEL
LIN {X 0,Y 601.383,Z 42.57,A -85,B 0,C 180,E1 -614.408,E2 -614.408} C_VEL
LIN {X 0,Y 601.409,Z 42.568,A -85,B 0,C 180,E1 -617.172,E2 -617.172} C_VEL
LIN {X 0,Y 601.416,Z 42.596,A -85,B 0,C 180,E1 -618.903,E2 -618.903} C_VEL
LIN {X 0,Y 601.414,Z 57.69,A -85,B 0,C 180,E1 -621.601,E2 -621.601} C_VEL
LIN {X 0,Y 601.379,Z 70.6,A -85,B 0,C 180,E1 -623.88,E2 -623.88} C_VEL
LIN {X 0,Y 601.645,Z 76.401,A -85,B 0,C 180,E1 -623.965,E2 -623.965} C_VEL
LIN {X 0,Y 601.574,Z 176.928,A -85,B 0,C 180,E1 -625.183,E2 -625.183} C_VEL
LIN {X 0,Y 601.573,Z 190.017,A -85,B 0,C 180,E1 -625.477,E2 -625.477} C_VEL
LIN {X 0,Y 601.538,Z 202.597,A -85,B 0,C 180,E1 -625.897,E2 -625.897} C_VEL
LIN {X 0,Y 601.516,Z 213.824,A -85,B 0,C 180,E1 -626.4,E2 -626.4} C_VEL
LIN {X 0,Y 601.486,Z 225.435,A -85,B 0,C 180,E1 -627.07,E2 -627.07} C_VEL
LIN {X 0,Y 601.431,Z 236.893,A -85,B 0,C 180,E1 -627.907,E2 -627.907} C_VEL
LIN {X 0,Y 601.416,Z 245.273,A -85,B 0,C 180,E1 -628.661,E2 -628.661} C_VEL
LIN {X 0,Y 601.393,Z 254.381,A -85,B 0,C 180,E1 -629.665,E2 -629.665} C_VEL
LIN {X 0,Y 601.366,Z 261.734,A -85,B 0,C 180,E1 -630.67,E2 -630.67} C_VEL
LIN {X 0,Y 601.359,Z 267.649,A -85,B 0,C 180,E1 -631.674,E2 -631.674} C_VEL
LIN {X 0,Y 601.335,Z 272.335,A -85,B 0,C 180,E1 -632.68,E2 -632.68} C_VEL
LIN {X 0,Y 601.367,Z 275.927,A -85,B 0,C 180,E1 -633.686,E2 -633.686} C_VEL
LIN {X 0,Y 601.328,Z 278.524,A -85,B 0,C 180,E1 -634.693,E2 -634.693} C_VEL
LIN {X 0,Y 601.336,Z 279.743,A -85,B 0,C 180,E1 -635.365,E2 -635.365} C_VEL
LIN {X 0,Y 601.35,Z 280.899,A -85,B 0,C 180,E1 -636.583,E2 -636.583} C_VEL
LIN {X 0,Y 601.322,Z 280.927,A -85,B 0,C 180,E1 -637.387,E2 -637.387} C_VEL
LIN {X 0,Y 601.332,Z 280.54,A -85,B 0,C 180,E1 -638.062,E2 -638.062} C_VEL
LIN {X 0,Y 601.333,Z 279.719,A -85,B 0,C 180,E1 -638.739,E2 -638.739} C_VEL
LIN {X 0,Y 601.336,Z 278.48,A -85,B 0,C 180,E1 -639.417,E2 -639.417} C_VEL
LIN {X 0,Y 601.355,Z 275.824,A -85,B 0,C 180,E1 -640.437,E2 -640.437} C_VEL
LIN {X 0,Y 601.332,Z 272.124,A -85,B 0,C 180,E1 -641.46,E2 -641.46} C_VEL
LIN {X 0,Y 601.38,Z 267.267,A -85,B 0,C 180,E1 -642.486,E2 -642.486} C_VEL
LIN {X 0,Y 601.37,Z 261.088,A -85,B 0,C 180,E1 -643.517,E2 -643.517} C_VEL
LIN {X 0,Y 601.405,Z 253.357,A -85,B 0,C 180,E1 -644.552,E2 -644.552} C_VEL
LIN {X 0,Y 601.425,Z 245.392,A -85,B 0,C 180,E1 -645.418,E2 -645.418} C_VEL
LIN {X 0,Y 601.465,Z 235.588,A -85,B 0,C 180,E1 -646.286,E2 -646.286} C_VEL
LIN {X 0,Y 601.468,Z 224.641,A -85,B 0,C 180,E1 -647.073,E2 -647.073} C_VEL
LIN {X 0,Y 601.502,Z 213.93,A -85,B 0,C 180,E1 -647.685,E2 -647.685} C_VEL
LIN {X 0,Y 601.548,Z 202.113,A -85,B 0,C 180,E1 -648.212,E2 -648.212} C_VEL
LIN {X 0,Y 601.604,Z 188.774,A -85,B 0,C 180,E1 -648.647,E2 -648.647} C_VEL
LIN {X 0,Y 601.631,Z 176.027,A -85,B 0,C 180,E1 -648.921,E2 -648.921} C_VEL
LIN {X 0,Y 601.554,Z 71.703,A -85,B 0,C 180,E1 -650.183,E2 -650.183} C_VEL
LIN {X 0,Y 601.405,Z 70.594,A -85,B 0,C 180,E1 -650.211,E2 -650.211} C_VEL
LIN {X 0,Y 601.455,Z 55.58,A -85,B 0,C 180,E1 -652.863,E2 -652.863} C_VEL
LIN {X 0,Y 601.381,Z 42.571,A -85,B 0,C 180,E1 -655.203,E2 -655.203} C_VEL
LIN {X 0,Y 601.371,Z 42.573,A -85,B 0,C 180,E1 -657.87,E2 -657.87} C_VEL
LIN {X 0,Y 601.407,Z 42.574,A -85,B 0,C 180,E1 -660.165,E2 -660.165} C_VEL
LIN {X 0,Y 601.401,Z 42.569,A -85,B 0,C 180,E1 -662.711,E2 -662.711} C_VEL
LIN {X 0,Y 601.354,Z 42.572,A -85,B 0,C 180,E1 -665.106,E2 -665.106} C_VEL
LIN {X 0,Y 601.385,Z 42.57,A -85,B 0,C 180,E1 -667.423,E2 -667.423} C_VEL
LIN {X 0,Y 601.377,Z 42.579,A -85,B 0,C 180,E1 -669.998,E2 -669.998} C_VEL
LIN {X 0,Y 601.347,Z 42.573,A -85,B 0,C 180,E1 -672.676,E2 -672.676} C_VEL
LIN {X 0,Y 601.404,Z 42.571,A -85,B 0,C 180,E1 -675.479,E2 -675.479} C_VEL
LIN {X 0,Y 601.373,Z 42.57,A -85,B 0,C 180,E1 -678.413,E2 -678.413} C_VEL
LIN {X 0,Y 601.368,Z 42.571,A -85,B 0,C 180,E1 -680.87,E2 -680.87} C_VEL
LIN {X 0,Y 601.384,Z 42.574,A -85,B 0,C 180,E1 -683.742,E2 -683.742} C_VEL
LIN {X 0,Y 601.373,Z 42.571,A -85,B 0,C 180,E1 -686.073,E2 -686.073} C_VEL
LIN {X 0,Y 601.386,Z 42.569,A -85,B 0,C 180,E1 -688.551,E2 -688.551} C_VEL
LIN {X 0,Y 601.421,Z 42.571,A -85,B 0,C 180,E1 -691.372,E2 -691.372} C_VEL
LIN {X 0,Y 601.357,Z 42.572,A -85,B 0,C 180,E1 -694.144,E2 -694.144} C_VEL
LIN {X 0,Y 601.367,Z 42.574,A -85,B 0,C 180,E1 -696.587,E2 -696.587} C_VEL
LIN {X 0,Y 601.403,Z 42.568,A -85,B 0,C 180,E1 -699.477,E2 -699.477} C_VEL
LIN {X 0,Y 601.372,Z 42.57,A -85,B 0,C 180,E1 -701.606,E2 -701.606} C_VEL
LIN {X 0,Y 601.401,Z 42.566,A -85,B 0,C 180,E1 -703.712,E2 -703.712} C_VEL
LIN {X 0,Y 601.406,Z 42.573,A -85,B 0,C 180,E1 -706.484,E2 -706.484} C_VEL
LIN {X 0,Y 601.388,Z 42.569,A -85,B 0,C 180,E1 -709.223,E2 -709.223} C_VEL
LIN {X 0,Y 601.396,Z 42.569,A -85,B 0,C 180,E1 -711.938,E2 -711.938} C_VEL
LIN {X 0,Y 601.423,Z 42.569,A -85,B 0,C 180,E1 -714.636,E2 -714.636} C_VEL
LIN {X 0,Y 601.405,Z 42.566,A -85,B 0,C 180,E1 -717.321,E2 -717.321} C_VEL
LIN {X 0,Y 601.438,Z 42.568,A -85,B 0,C 180,E1 -720,E2 -720} C_VEL
LIN {X 0,Y 601.43,Z 42.564,A -85,B 0,C 180,E1 -722.679,E2 -722.679} C_VEL
LIN {X 0,Y 601.397,Z 42.568,A -85,B 0,C 180,E1 -725.364,E2 -725.364} C_VEL
LIN {X 0,Y 601.437,Z 42.569,A -85,B 0,C 180,E1 -728.061,E2 -728.061} C_VEL
LIN {X 0,Y 601.394,Z 42.567,A -85,B 0,C 180,E1 -730.995,E2 -730.995} C_VEL
LIN {X 0,Y 601.404,Z 42.573,A -85,B 0,C 180,E1 -733.516,E2 -733.516} C_VEL
LIN {X 0,Y 601.416,Z 42.565,A -85,B 0,C 180,E1 -736.287,E2 -736.287} C_VEL
LIN {X 0,Y 601.41,Z 42.569,A -85,B 0,C 180,E1 -739.099,E2 -739.099} C_VEL
LIN {X 0,Y 601.402,Z 42.568,A -85,B 0,C 180,E1 -741.96,E2 -741.96} C_VEL
LIN {X 0,Y 601.393,Z 42.571,A -85,B 0,C 180,E1 -744.879,E2 -744.879} C_VEL
LIN {X 0,Y 601.416,Z 42.572,A -85,B 0,C 180,E1 -747.362,E2 -747.362} C_VEL
LIN {X 0,Y 601.404,Z 42.566,A -85,B 0,C 180,E1 -750.165,E2 -750.165} C_VEL
LIN {X 0,Y 601.407,Z 42.571,A -85,B 0,C 180,E1 -752.713,E2 -752.713} C_VEL
LIN {X 0,Y 601.399,Z 42.573,A -85,B 0,C 180,E1 -755.112,E2 -755.112} C_VEL
LIN {X 0,Y 601.436,Z 42.563,A -85,B 0,C 180,E1 -757.419,E2 -757.419} C_VEL
LIN {X 0,Y 601.403,Z 42.567,A -85,B 0,C 180,E1 -759.996,E2 -759.996} C_VEL
LIN {X 0,Y 601.41,Z 42.575,A -85,B 0,C 180,E1 -762.671,E2 -762.671} C_VEL
LIN {X 0,Y 601.401,Z 42.566,A -85,B 0,C 180,E1 -765.479,E2 -765.479} C_VEL
LIN {X 0,Y 601.424,Z 42.573,A -85,B 0,C 180,E1 -768.407,E2 -768.407} C_VEL
LIN {X 0,Y 601.432,Z 42.565,A -85,B 0,C 180,E1 -770.875,E2 -770.875} C_VEL
LIN {X 0,Y 601.404,Z 42.566,A -85,B 0,C 180,E1 -773.417,E2 -773.417} C_VEL
LIN {X 0,Y 601.434,Z 42.57,A -85,B 0,C 180,E1 -776.064,E2 -776.064} C_VEL
LIN {X 0,Y 601.415,Z 42.565,A -85,B 0,C 180,E1 -779.057,E2 -779.057} C_VEL
LIN {X 0,Y 601.419,Z 42.566,A -85,B 0,C 180,E1 -781.372,E2 -781.372} C_VEL
LIN {X 0,Y 601.398,Z 42.572,A -85,B 0,C 180,E1 -783.636,E2 -783.636} C_VEL
LIN {X 0,Y 601.425,Z 42.567,A -85,B 0,C 180,E1 -786.59,E2 -786.59} C_VEL
LIN {X 0,Y 601.454,Z 42.815,A -85,B 0,C 180,E1 -786.773,E2 -786.773} C_VEL
LIN {X 0,Y 601.703,Z 47.69,A -85,B 0,C 180,E1 -787.449,E2 -787.449} C_VEL
LIN {X 0,Y 601.58,Z 66.748,A -85,B 0,C 180,E1 -790.018,E2 -790.018} C_VEL
LIN {X 0,Y 601.547,Z 86.692,A -85,B 0,C 180,E1 -792.667,E2 -792.667} C_VEL
LIN {X 0,Y 601.467,Z 106.636,A -85,B 0,C 180,E1 -795.277,E2 -795.277} C_VEL
LIN {X 0,Y 601.425,Z 118.52,A -85,B 0,C 180,E1 -796.817,E2 -796.817} C_VEL
LIN {X 0,Y 601.638,Z 131.644,A -85,B 0,C 180,E1 -796.983,E2 -796.983} C_VEL
LIN {X 0,Y 601.623,Z 226.934,A -85,B 0,C 180,E1 -798.14,E2 -798.14} C_VEL
LIN {X 0,Y 601.562,Z 240.209,A -85,B 0,C 180,E1 -798.437,E2 -798.437} C_VEL
LIN {X 0,Y 601.544,Z 252.629,A -85,B 0,C 180,E1 -798.853,E2 -798.853} C_VEL
LIN {X 0,Y 601.522,Z 264.628,A -85,B 0,C 180,E1 -799.396,E2 -799.396} C_VEL
LIN {X 0,Y 601.479,Z 276.196,A -85,B 0,C 180,E1 -800.075,E2 -800.075} C_VEL
LIN {X 0,Y 601.444,Z 286.593,A -85,B 0,C 180,E1 -800.839,E2 -800.839} C_VEL
LIN {X 0,Y 601.429,Z 295.11,A -85,B 0,C 180,E1 -801.601,E2 -801.601} C_VEL
LIN {X 0,Y 601.418,Z 302.959,A -85,B 0,C 180,E1 -802.446,E2 -802.446} C_VEL
LIN {X 0,Y 601.37,Z 310.224,A -85,B 0,C 180,E1 -803.398,E2 -803.398} C_VEL
LIN {X 0,Y 601.372,Z 315.865,A -85,B 0,C 180,E1 -804.299,E2 -804.299} C_VEL
LIN {X 0,Y 601.336,Z 320.949,A -85,B 0,C 180,E1 -805.307,E2 -805.307} C_VEL
LIN {X 0,Y 601.368,Z 324.895,A -85,B 0,C 180,E1 -806.314,E2 -806.314} C_VEL
LIN {X 0,Y 601.325,Z 327.808,A -85,B 0,C 180,E1 -807.32,E2 -807.32} C_VEL
LIN {X 0,Y 601.343,Z 329.201,A -85,B 0,C 180,E1 -807.991,E2 -807.991} C_VEL
LIN {X 0,Y 601.339,Z 330.784,A -85,B 0,C 180,E1 -809.33,E2 -809.33} C_VEL
LIN {X 0,Y 601.335,Z 331,A -85,B 0,C 180,E1 -810,E2 -810} C_VEL
LIN {X 0,Y 601.347,Z 330.185,A -85,B 0,C 180,E1 -811.339,E2 -811.339} C_VEL
LIN {X 0,Y 601.343,Z 329.202,A -85,B 0,C 180,E1 -812.009,E2 -812.009} C_VEL
LIN {X 0,Y 601.325,Z 327.81,A -85,B 0,C 180,E1 -812.679,E2 -812.679} C_VEL
LIN {X 0,Y 601.368,Z 324.897,A -85,B 0,C 180,E1 -813.685,E2 -813.685} C_VEL
LIN {X 0,Y 601.336,Z 320.95,A -85,B 0,C 180,E1 -814.692,E2 -814.692} C_VEL
LIN {X 0,Y 601.373,Z 314.878,A -85,B 0,C 180,E1 -815.869,E2 -815.869} C_VEL
LIN {X 0,Y 601.381,Z 308.237,A -85,B 0,C 180,E1 -816.88,E2 -816.88} C_VEL
LIN {X 0,Y 601.4,Z 299.991,A -85,B 0,C 180,E1 -817.892,E2 -817.892} C_VEL
LIN {X 0,Y 601.436,Z 291.539,A -85,B 0,C 180,E1 -818.737,E2 -818.737} C_VEL
LIN {X 0,Y 601.448,Z 281.096,A -85,B 0,C 180,E1 -819.585,E2 -819.585} C_VEL
LIN {X 0,Y 601.465,Z 270.762,A -85,B 0,C 180,E1 -820.264,E2 -820.264} C_VEL
LIN {X 0,Y 601.538,Z 258.595,A -85,B 0,C 180,E1 -820.896,E2 -820.896} C_VEL
LIN {X 0,Y 601.556,Z 246.222,A -85,B 0,C 180,E1 -821.379,E2 -821.379} C_VEL
LIN {X 0,Y 601.585,Z 233.445,A -85,B 0,C 180,E1 -821.733,E2 -821.733} C_VEL
LIN {X 0,Y 601.625,Z 221.098,A -85,B 0,C 180,E1 -821.946,E2 -821.946} C_VEL
LIN {X 0,Y 601.505,Z 119.157,A -85,B 0,C 180,E1 -823.17,E2 -823.17} C_VEL
LIN {X 0,Y 601.444,Z 118.274,A -85,B 0,C 180,E1 -823.214,E2 -823.214} C_VEL
LIN {X 0,Y 601.513,Z 96.003,A -85,B 0,C 180,E1 -826.11,E2 -826.11} C_VEL
LIN {X 0,Y 601.532,Z 76.092,A -85,B 0,C 180,E1 -828.737,E2 -828.737} C_VEL
LIN {X 0,Y 601.672,Z 54.785,A -85,B 0,C 180,E1 -831.589,E2 -831.589} C_VEL
LIN {X 0,Y 601.685,Z 44.148,A -85,B 0,C 180,E1 -833.035,E2 -833.035} C_VEL
LIN {X 0,Y 601.413,Z 42.569,A -85,B 0,C 180,E1 -833.274,E2 -833.274} C_VEL
LIN {X 0,Y 601.41,Z 42.572,A -85,B 0,C 180,E1 -835.866,E2 -835.866} C_VEL
LIN {X 0,Y 601.402,Z 42.573,A -85,B 0,C 180,E1 -837.868,E2 -837.868} C_VEL
LIN {X 0,Y 601.43,Z 42.57,A -85,B 0,C 180,E1 -840.164,E2 -840.164} C_VEL
LIN {X 0,Y 601.412,Z 42.565,A -85,B 0,C 180,E1 -842.714,E2 -842.714} C_VEL
LIN {X 0,Y 601.397,Z 42.567,A -85,B 0,C 180,E1 -845.112,E2 -845.112} C_VEL
LIN {X 0,Y 601.436,Z 42.567,A -85,B 0,C 180,E1 -847.419,E2 -847.419} C_VEL
LIN {X 0,Y 601.413,Z 42.569,A -85,B 0,C 180,E1 -849.995,E2 -849.995} C_VEL
LIN {X 0,Y 601.408,Z 42.565,A -85,B 0,C 180,E1 -852.67,E2 -852.67} C_VEL
LIN {X 0,Y 601.398,Z 42.577,A -85,B 0,C 180,E1 -855.479,E2 -855.479} C_VEL
LIN {X 0,Y 601.421,Z 42.564,A -85,B 0,C 180,E1 -858.407,E2 -858.407} C_VEL
LIN {X 0,Y 601.406,Z 42.569,A -85,B 0,C 180,E1 -860.873,E2 -860.873} C_VEL
LIN {X 0,Y 601.401,Z 42.574,A -85,B 0,C 180,E1 -863.417,E2 -863.417} C_VEL
LIN {X 0,Y 601.432,Z 42.562,A -85,B 0,C 180,E1 -866.064,E2 -866.064} C_VEL
LIN {X 0,Y 601.421,Z 42.574,A -85,B 0,C 180,E1 -869.058,E2 -869.058} C_VEL
LIN {X 0,Y 601.419,Z 42.568,A -85,B 0,C 180,E1 -871.372,E2 -871.372} C_VEL
LIN {X 0,Y 601.399,Z 42.567,A -85,B 0,C 180,E1 -873.636,E2 -873.636} C_VEL
LIN {X 0,Y 601.447,Z 42.56,A -85,B 0,C 180,E1 -875.859,E2 -875.859} C_VEL
LIN {X 0,Y 601.402,Z 42.577,A -85,B 0,C 180,E1 -878.761,E2 -878.761} C_VEL
LIN {X 0,Y 601.413,Z 42.565,A -85,B 0,C 180,E1 -881.608,E2 -881.608} C_VEL
LIN {X 0,Y 601.412,Z 42.572,A -85,B 0,C 180,E1 -884.409,E2 -884.409} C_VEL
LIN {X 0,Y 601.407,Z 42.567,A -85,B 0,C 180,E1 -887.172,E2 -887.172} C_VEL
LIN {X 0,Y 601.432,Z 42.565,A -85,B 0,C 180,E1 -889.905,E2 -889.905} C_VEL
LIN {X 0,Y 601.403,Z 42.571,A -85,B 0,C 180,E1 -892.615,E2 -892.615} C_VEL
LIN {X 0,Y 601.413,Z 42.565,A -85,B 0,C 180,E1 -895.308,E2 -895.308} C_VEL
LIN {X 0,Y 601.433,Z 42.57,A -85,B 0,C 180,E1 -897.991,E2 -897.991} C_VEL
LIN {X 0,Y 601.429,Z 42.564,A -85,B 0,C 180,E1 -900.67,E2 -900.67} C_VEL
LIN {X 0,Y 601.426,Z 42.564,A -85,B 0,C 180,E1 -903.35,E2 -903.35} C_VEL
LIN {X 0,Y 601.415,Z 42.572,A -85,B 0,C 180,E1 -906.037,E2 -906.037} C_VEL
LIN {X 0,Y 601.4,Z 42.566,A -85,B 0,C 180,E1 -908.738,E2 -908.738} C_VEL
LIN {X 0,Y 601.437,Z 42.567,A -85,B 0,C 180,E1 -911.458,E2 -911.458} C_VEL
LIN {X 0,Y 601.398,Z 42.568,A -85,B 0,C 180,E1 -912.348,E2 -912.348} C_VEL
LIN {X 0,Y 600.727,Z 42.651,A -85,B 0,C 180,E1 -912.907,E2 -912.907} C_VEL
LIN {X 0,Y 597.873,Z 43.013,A -85,B 0,C 180,E1 -913.815,E2 -913.815} C_VEL
LIN {X 0,Y 595.464,Z 43.31,A -85,B 0,C 180,E1 -914.545,E2 -914.545} C_VEL
LIN {X 0,Y 594.43,Z 43.437,A -85,B 0,C 180,E1 -915.109,E2 -915.109} C_VEL
LIN {X 0,Y 594.346,Z 43.447,A -85,B 0,C 180,E1 -915.299,E2 -915.299} C_VEL
LIN {X 0,Y 594.339,Z 43.45,A -85,B 0,C 180,E1 -917.906,E2 -917.906} C_VEL
LIN {X 0,Y 594.395,Z 43.44,A -85,B 0,C 180,E1 -920.776,E2 -920.776} C_VEL
LIN {X 0,Y 594.365,Z 43.447,A -85,B 0,C 180,E1 -923.705,E2 -923.705} C_VEL
LIN {X 0,Y 594.381,Z 43.443,A -85,B 0,C 180,E1 -926.7,E2 -926.7} C_VEL
LIN {X 0,Y 594.378,Z 43.448,A -85,B 0,C 180,E1 -928.999,E2 -928.999} C_VEL
LIN {X 0,Y 594.371,Z 43.444,A -85,B 0,C 180,E1 -931.642,E2 -931.642} C_VEL
LIN {X 0,Y 594.377,Z 43.445,A -85,B 0,C 180,E1 -934.581,E2 -934.581} C_VEL
LIN {X 0,Y 594.384,Z 43.441,A -85,B 0,C 180,E1 -937.608,E2 -937.608} C_VEL
LIN {X 0,Y 594.361,Z 43.449,A -85,B 0,C 180,E1 -940.568,E2 -940.568} C_VEL
LIN {X 0,Y 594.351,Z 43.446,A -85,B 0,C 180,E1 -943.301,E2 -943.301} C_VEL
LIN {X 0,Y 594.362,Z 43.446,A -85,B 0,C 180,E1 -946.162,E2 -946.162} C_VEL
LIN {X 0,Y 594.366,Z 43.444,A -85,B 0,C 180,E1 -949.18,E2 -949.18} C_VEL
LIN {X 0,Y 594.369,Z 43.446,A -85,B 0,C 180,E1 -952.058,E2 -952.058} C_VEL
LIN {X 0,Y 594.327,Z 43.452,A -85,B 0,C 180,E1 -954.681,E2 -954.681} C_VEL
LIN {X 0,Y 594.374,Z 43.442,A -85,B 0,C 180,E1 -957.09,E2 -957.09} C_VEL
LIN {X 0,Y 594.388,Z 43.442,A -85,B 0,C 180,E1 -959.673,E2 -959.673} C_VEL
LIN {X 0,Y 594.336,Z 43.45,A -85,B 0,C 180,E1 -962.537,E2 -962.537} C_VEL
LIN {X 0,Y 594.332,Z 43.447,A -85,B 0,C 180,E1 -964.805,E2 -964.805} C_VEL
LIN {X 0,Y 594.361,Z 43.444,A -85,B 0,C 180,E1 -967.267,E2 -967.267} C_VEL
LIN {X 0,Y 594.366,Z 43.452,A -85,B 0,C 180,E1 -969.946,E2 -969.946} C_VEL
LIN {X 0,Y 594.343,Z 43.445,A -85,B 0,C 180,E1 -972.805,E2 -972.805} C_VEL
LIN {X 0,Y 594.367,Z 43.451,A -85,B 0,C 180,E1 -975.837,E2 -975.837} C_VEL
LIN {X 0,Y 594.355,Z 43.446,A -85,B 0,C 180,E1 -978.761,E2 -978.761} C_VEL
LIN {X 0,Y 594.433,Z 43.837,A -85,B 0,C 180,E1 -978.908,E2 -978.908} C_VEL
LIN {X 0,Y 594.403,Z 58.174,A -85,B 0,C 180,E1 -981.501,E2 -981.501} C_VEL
LIN {X 0,Y 594.349,Z 70.791,A -85,B 0,C 180,E1 -983.734,E2 -983.734} C_VEL
LIN {X 0,Y 594.743,Z 74.708,A -85,B 0,C 180,E1 -983.79,E2 -983.79} C_VEL
LIN {X 0,Y 594.636,Z 176.883,A -85,B 0,C 180,E1 -985.042,E2 -985.042} C_VEL
LIN {X 0,Y 594.617,Z 189.991,A -85,B 0,C 180,E1 -985.339,E2 -985.339} C_VEL
LIN {X 0,Y 594.576,Z 202.578,A -85,B 0,C 180,E1 -985.764,E2 -985.764} C_VEL
LIN {X 0,Y 594.543,Z 213.812,A -85,B 0,C 180,E1 -986.273,E2 -986.273} C_VEL
LIN {X 0,Y 594.475,Z 225.425,A -85,B 0,C 180,E1 -986.951,E2 -986.951} C_VEL
LIN {X 0,Y 594.395,Z 236.89,A -85,B 0,C 180,E1 -987.798,E2 -987.798} C_VEL
LIN {X 0,Y 594.373,Z 246.108,A -85,B 0,C 180,E1 -988.645,E2 -988.645} C_VEL
LIN {X 0,Y 594.322,Z 255.053,A -85,B 0,C 180,E1 -989.661,E2 -989.661} C_VEL
LIN {X 0,Y 594.295,Z 262.285,A -85,B 0,C 180,E1 -990.678,E2 -990.678} C_VEL
LIN {X 0,Y 594.28,Z 268.096,A -85,B 0,C 180,E1 -991.694,E2 -991.694} C_VEL
LIN {X 0,Y 594.24,Z 272.688,A -85,B 0,C 180,E1 -992.712,E2 -992.712} C_VEL
LIN {X 0,Y 594.269,Z 275.131,A -85,B 0,C 180,E1 -993.39,E2 -993.39} C_VEL
LIN {X 0,Y 594.255,Z 277.123,A -85,B 0,C 180,E1 -994.069,E2 -994.069} C_VEL
LIN {X 0,Y 594.227,Z 278.703,A -85,B 0,C 180,E1 -994.749,E2 -994.749} C_VEL
LIN {X 0,Y 594.251,Z 279.875,A -85,B 0,C 180,E1 -995.429,E2 -995.429} C_VEL
LIN {X 0,Y 594.272,Z 280.948,A -85,B 0,C 180,E1 -996.792,E2 -996.792} C_VEL
LIN {X 0,Y 594.248,Z 280.907,A -85,B 0,C 180,E1 -997.475,E2 -997.475} C_VEL
LIN {X 0,Y 594.228,Z 280.462,A -85,B 0,C 180,E1 -998.159,E2 -998.159} C_VEL
LIN {X 0,Y 594.256,Z 278.301,A -85,B 0,C 180,E1 -999.531,E2 -999.531} C_VEL
LIN {X 0,Y 594.281,Z 275.559,A -85,B 0,C 180,E1 -1000.562,E2 -1000.562} C_VEL
LIN {X 0,Y 594.248,Z 271.766,A -85,B 0,C 180,E1 -1001.599,E2 -1001.599} C_VEL
LIN {X 0,Y 594.286,Z 266.808,A -85,B 0,C 180,E1 -1002.638,E2 -1002.638} C_VEL
LIN {X 0,Y 594.296,Z 260.52,A -85,B 0,C 180,E1 -1003.681,E2 -1003.681} C_VEL
LIN {X 0,Y 594.334,Z 252.626,A -85,B 0,C 180,E1 -1004.729,E2 -1004.729} C_VEL
LIN {X 0,Y 594.362,Z 244.484,A -85,B 0,C 180,E1 -1005.605,E2 -1005.605} C_VEL
LIN {X 0,Y 594.416,Z 234.499,A -85,B 0,C 180,E1 -1006.485,E2 -1006.485} C_VEL
LIN {X 0,Y 594.445,Z 223.245,A -85,B 0,C 180,E1 -1007.281,E2 -1007.281} C_VEL
LIN {X 0,Y 594.531,Z 212.147,A -85,B 0,C 180,E1 -1007.9,E2 -1007.9} C_VEL
LIN {X 0,Y 594.602,Z 199.817,A -85,B 0,C 180,E1 -1008.432,E2 -1008.432} C_VEL
LIN {X 0,Y 594.615,Z 187.162,A -85,B 0,C 180,E1 -1008.829,E2 -1008.829} C_VEL
LIN {X 0,Y 594.674,Z 173.516,A -85,B 0,C 180,E1 -1009.098,E2 -1009.098} C_VEL
LIN {X 0,Y 594.627,Z 72.321,A -85,B 0,C 180,E1 -1010.331,E2 -1010.331} C_VEL
LIN {X 0,Y 594.384,Z 70.591,A -85,B 0,C 180,E1 -1010.369,E2 -1010.369} C_VEL
LIN {X 0,Y 594.409,Z 54.035,A -85,B 0,C 180,E1 -1013.334,E2 -1013.334} C_VEL
LIN {X 0,Y 594.367,Z 43.783,A -85,B 0,C 180,E1 -1015.194,E2 -1015.194} C_VEL
LIN {X 0,Y 594.335,Z 43.45,A -85,B 0,C 180,E1 -1015.289,E2 -1015.289} C_VEL
LIN {X 0,Y 594.329,Z 43.448,A -85,B 0,C 180,E1 -1017.515,E2 -1017.515} C_VEL
LIN {X 0,Y 594.369,Z 43.452,A -85,B 0,C 180,E1 -1020.324,E2 -1020.324} C_VEL
LIN {X 0,Y 594.341,Z 43.447,A -85,B 0,C 180,E1 -1022.953,E2 -1022.953} C_VEL
LIN {X 0,Y 594.31,Z 43.451,A -85,B 0,C 180,E1 -1025.412,E2 -1025.412} C_VEL
LIN {X 0,Y 594.349,Z 43.454,A -85,B 0,C 180,E1 -1027.944,E2 -1027.944} C_VEL
LIN {X 0,Y 594.328,Z 43.448,A -85,B 0,C 180,E1 -1030.816,E2 -1030.816} C_VEL
LIN {X 0,Y 594.336,Z 43.449,A -85,B 0,C 180,E1 -1033.303,E2 -1033.303} C_VEL
LIN {X 0,Y 594.343,Z 43.449,A -85,B 0,C 180,E1 -1036.163,E2 -1036.163} C_VEL
LIN {X 0,Y 594.333,Z 43.447,A -85,B 0,C 180,E1 -1038.532,E2 -1038.532} C_VEL
LIN {X 0,Y 594.324,Z 43.454,A -85,B 0,C 180,E1 -1041.303,E2 -1041.303} C_VEL
LIN {X 0,Y 594.338,Z 43.451,A -85,B 0,C 180,E1 -1043.754,E2 -1043.754} C_VEL
LIN {X 0,Y 594.321,Z 43.449,A -85,B 0,C 180,E1 -1046.235,E2 -1046.235} C_VEL
LIN {X 0,Y 594.338,Z 43.447,A -85,B 0,C 180,E1 -1048.647,E2 -1048.647} C_VEL
LIN {X 0,Y 594.377,Z 43.449,A -85,B 0,C 180,E1 -1051.044,E2 -1051.044} C_VEL
LIN {X 0,Y 594.324,Z 43.448,A -85,B 0,C 180,E1 -1054.053,E2 -1054.053} C_VEL
LIN {X 0,Y 594.336,Z 43.447,A -85,B 0,C 180,E1 -1056.293,E2 -1056.293} C_VEL
LIN {X 0,Y 594.389,Z 43.445,A -85,B 0,C 180,E1 -1059.224,E2 -1059.224} C_VEL
LIN {X 0,Y 594.325,Z 43.448,A -85,B 0,C 180,E1 -1062.094,E2 -1062.094} C_VEL
LIN {X 0,Y 594.342,Z 43.448,A -85,B 0,C 180,E1 -1064.218,E2 -1064.218} C_VEL
LIN {X 0,Y 594.33,Z 43.451,A -85,B 0,C 180,E1 -1067.016,E2 -1067.016} C_VEL
LIN {X 0,Y 594.354,Z 43.446,A -85,B 0,C 180,E1 -1069.094,E2 -1069.094} C_VEL
LIN {X 0,Y 594.349,Z 43.446,A -85,B 0,C 180,E1 -1071.842,E2 -1071.842} C_VEL
LIN {X 0,Y 594.385,Z 43.447,A -85,B 0,C 180,E1 -1074.572,E2 -1074.572} C_VEL
LIN {X 0,Y 594.376,Z 43.441,A -85,B 0,C 180,E1 -1077.289,E2 -1077.289} C_VEL
LIN {X 0,Y 594.407,Z 43.444,A -85,B 0,C 180,E1 -1080,E2 -1080} C_VEL
LIN {X 0,Y 594.394,Z 43.441,A -85,B 0,C 180,E1 -1082.711,E2 -1082.711} C_VEL
LIN {X 0,Y 594.366,Z 43.444,A -85,B 0,C 180,E1 -1085.428,E2 -1085.428} C_VEL
LIN {X 0,Y 594.381,Z 43.446,A -85,B 0,C 180,E1 -1088.157,E2 -1088.157} C_VEL
LIN {X 0,Y 594.367,Z 43.443,A -85,B 0,C 180,E1 -1091.061,E2 -1091.061} C_VEL
LIN {X 0,Y 594.374,Z 43.451,A -85,B 0,C 180,E1 -1093.679,E2 -1093.679} C_VEL
LIN {X 0,Y 594.346,Z 43.445,A -85,B 0,C 180,E1 -1096.702,E2 -1096.702} C_VEL
LIN {X 0,Y 594.362,Z 43.45,A -85,B 0,C 180,E1 -1099.335,E2 -1099.335} C_VEL
LIN {X 0,Y 594.36,Z 43.451,A -85,B 0,C 180,E1 -1101.504,E2 -1101.504} C_VEL
LIN {X 0,Y 594.369,Z 43.442,A -85,B 0,C 180,E1 -1104.447,E2 -1104.447} C_VEL
LIN {X 0,Y 594.371,Z 43.444,A -85,B 0,C 180,E1 -1106.7,E2 -1106.7} C_VEL
LIN {X 0,Y 594.376,Z 43.449,A -85,B 0,C 180,E1 -1108.999,E2 -1108.999} C_VEL
LIN {X 0,Y 594.376,Z 43.443,A -85,B 0,C 180,E1 -1111.642,E2 -1111.642} C_VEL
LIN {X 0,Y 594.381,Z 43.445,A -85,B 0,C 180,E1 -1114.58,E2 -1114.58} C_VEL
LIN {X 0,Y 594.388,Z 43.44,A -85,B 0,C 180,E1 -1117.608,E2 -1117.608} C_VEL
LIN {X 0,Y 594.363,Z 43.45,A -85,B 0,C 180,E1 -1120.568,E2 -1120.568} C_VEL
LIN {X 0,Y 594.369,Z 43.444,A -85,B 0,C 180,E1 -1123.299,E2 -1123.299} C_VEL
LIN {X 0,Y 594.362,Z 43.447,A -85,B 0,C 180,E1 -1126.161,E2 -1126.161} C_VEL
LIN {X 0,Y 594.382,Z 43.449,A -85,B 0,C 180,E1 -1128.536,E2 -1128.536} C_VEL
LIN {X 0,Y 594.38,Z 43.441,A -85,B 0,C 180,E1 -1131.296,E2 -1131.296} C_VEL
LIN {X 0,Y 594.353,Z 43.447,A -85,B 0,C 180,E1 -1133.755,E2 -1133.755} C_VEL
LIN {X 0,Y 594.378,Z 43.451,A -85,B 0,C 180,E1 -1136.238,E2 -1136.238} C_VEL
LIN {X 0,Y 594.373,Z 43.445,A -85,B 0,C 180,E1 -1138.65,E2 -1138.65} C_VEL
LIN {X 0,Y 594.38,Z 43.442,A -85,B 0,C 180,E1 -1141.043,E2 -1141.043} C_VEL
LIN {X 0,Y 594.383,Z 43.442,A -85,B 0,C 180,E1 -1143.3,E2 -1143.3} C_VEL
LIN {X 0,Y 594.394,Z 43.445,A -85,B 0,C 180,E1 -1146.296,E2 -1146.296} C_VEL
LIN {X 0,Y 594.391,Z 43.573,A -85,B 0,C 180,E1 -1146.619,E2 -1146.619} C_VEL
LIN {X 0,Y 594.761,Z 48.39,A -85,B 0,C 180,E1 -1147.283,E2 -1147.283} C_VEL
LIN {X 0,Y 594.669,Z 66.748,A -85,B 0,C 180,E1 -1149.776,E2 -1149.776} C_VEL
LIN {X 0,Y 594.578,Z 88.022,A -85,B 0,C 180,E1 -1152.635,E2 -1152.635} C_VEL
LIN {X 0,Y 594.448,Z 107.966,A -85,B 0,C 180,E1 -1155.274,E2 -1155.274} C_VEL
LIN {X 0,Y 594.434,Z 118.437,A -85,B 0,C 180,E1 -1156.649,E2 -1156.649} C_VEL
LIN {X 0,Y 594.75,Z 124.489,A -85,B 0,C 180,E1 -1156.743,E2 -1156.743} C_VEL
LIN {X 0,Y 594.693,Z 226.934,A -85,B 0,C 180,E1 -1157.999,E2 -1157.999} C_VEL
LIN {X 0,Y 594.604,Z 240.211,A -85,B 0,C 180,E1 -1158.3,E2 -1158.3} C_VEL
LIN {X 0,Y 594.599,Z 252.423,A -85,B 0,C 180,E1 -1158.713,E2 -1158.713} C_VEL
LIN {X 0,Y 594.536,Z 264.627,A -85,B 0,C 180,E1 -1159.27,E2 -1159.27} C_VEL
LIN {X 0,Y 594.474,Z 276.198,A -85,B 0,C 180,E1 -1159.957,E2 -1159.957} C_VEL
LIN {X 0,Y 594.414,Z 286.595,A -85,B 0,C 180,E1 -1160.729,E2 -1160.729} C_VEL
LIN {X 0,Y 594.383,Z 295.11,A -85,B 0,C 180,E1 -1161.5,E2 -1161.5} C_VEL
LIN {X 0,Y 594.347,Z 302.959,A -85,B 0,C 180,E1 -1162.355,E2 -1162.355} C_VEL
LIN {X 0,Y 594.283,Z 310.812,A -85,B 0,C 180,E1 -1163.408,E2 -1163.408} C_VEL
LIN {X 0,Y 594.289,Z 317.679,A -85,B 0,C 180,E1 -1164.571,E2 -1164.571} C_VEL
LIN {X 0,Y 594.27,Z 322.371,A -85,B 0,C 180,E1 -1165.591,E2 -1165.591} C_VEL
LIN {X 0,Y 594.267,Z 325.956,A -85,B 0,C 180,E1 -1166.61,E2 -1166.61} C_VEL
LIN {X 0,Y 594.226,Z 327.808,A -85,B 0,C 180,E1 -1167.288,E2 -1167.288} C_VEL
LIN {X 0,Y 594.242,Z 329.2,A -85,B 0,C 180,E1 -1167.966,E2 -1167.966} C_VEL
LIN {X 0,Y 594.239,Z 330.784,A -85,B 0,C 180,E1 -1169.322,E2 -1169.322} C_VEL
LIN {X 0,Y 594.236,Z 331,A -85,B 0,C 180,E1 -1170,E2 -1170} C_VEL
LIN {X 0,Y 594.247,Z 330.185,A -85,B 0,C 180,E1 -1171.355,E2 -1171.355} C_VEL
LIN {X 0,Y 594.242,Z 329.201,A -85,B 0,C 180,E1 -1172.033,E2 -1172.033} C_VEL
LIN {X 0,Y 594.226,Z 327.81,A -85,B 0,C 180,E1 -1172.711,E2 -1172.711} C_VEL
LIN {X 0,Y 594.289,Z 324.897,A -85,B 0,C 180,E1 -1173.729,E2 -1173.729} C_VEL
LIN {X 0,Y 594.241,Z 320.95,A -85,B 0,C 180,E1 -1174.749,E2 -1174.749} C_VEL
LIN {X 0,Y 594.305,Z 314.879,A -85,B 0,C 180,E1 -1175.939,E2 -1175.939} C_VEL
LIN {X 0,Y 594.308,Z 308.238,A -85,B 0,C 180,E1 -1176.962,E2 -1176.962} C_VEL
LIN {X 0,Y 594.359,Z 299.992,A -85,B 0,C 180,E1 -1177.986,E2 -1177.986} C_VEL
LIN {X 0,Y 594.382,Z 291.54,A -85,B 0,C 180,E1 -1178.842,E2 -1178.842} C_VEL
LIN {X 0,Y 594.43,Z 281.098,A -85,B 0,C 180,E1 -1179.699,E2 -1179.699} C_VEL
LIN {X 0,Y 594.472,Z 270.761,A -85,B 0,C 180,E1 -1180.386,E2 -1180.386} C_VEL
LIN {X 0,Y 594.558,Z 259.722,A -85,B 0,C 180,E1 -1180.973,E2 -1180.973} C_VEL
LIN {X 0,Y 594.58,Z 247.715,A -85,B 0,C 180,E1 -1181.464,E2 -1181.464} C_VEL
LIN {X 0,Y 594.635,Z 234.358,A -85,B 0,C 180,E1 -1181.85,E2 -1181.85} C_VEL
LIN {X 0,Y 594.697,Z 221.098,A -85,B 0,C 180,E1 -1182.087,E2 -1182.087} C_VEL
LIN {X 0,Y 594.621,Z 120.052,A -85,B 0,C 180,E1 -1183.314,E2 -1183.314} C_VEL
LIN {X 0,Y 594.415,Z 118.274,A -85,B 0,C 180,E1 -1183.373,E2 -1183.373} C_VEL
LIN {X 0,Y 594.535,Z 96.003,A -85,B 0,C 180,E1 -1186.305,E2 -1186.305} C_VEL
LIN {X 0,Y 594.583,Z 76.785,A -85,B 0,C 180,E1 -1188.871,E2 -1188.871} C_VEL
LIN {X 0,Y 594.767,Z 56.114,A -85,B 0,C 180,E1 -1191.67,E2 -1191.67} C_VEL
LIN {X 0,Y 594.708,Z 45.291,A -85,B 0,C 180,E1 -1193.137,E2 -1193.137} C_VEL
LIN {X 0,Y 594.392,Z 43.445,A -85,B 0,C 180,E1 -1193.427,E2 -1193.427} C_VEL
LIN {X 0,Y 594.384,Z 43.45,A -85,B 0,C 180,E1 -1196.022,E2 -1196.022} C_VEL
LIN {X 0,Y 594.382,Z 43.441,A -85,B 0,C 180,E1 -1198.957,E2 -1198.957} C_VEL
LIN {X 0,Y 594.384,Z 43.446,A -85,B 0,C 180,E1 -1201.643,E2 -1201.643} C_VEL
LIN {X 0,Y 594.38,Z 43.441,A -85,B 0,C 180,E1 -1204.58,E2 -1204.58} C_VEL
LIN {X 0,Y 594.39,Z 43.447,A -85,B 0,C 180,E1 -1207.608,E2 -1207.608} C_VEL
LIN {X 0,Y 594.378,Z 43.45,A -85,B 0,C 180,E1 -1209.774,E2 -1209.774} C_VEL
LIN {X 0,Y 594.364,Z 43.443,A -85,B 0,C 180,E1 -1212.376,E2 -1212.376} C_VEL
LIN {X 0,Y 594.336,Z 43.451,A -85,B 0,C 180,E1 -1215.194,E2 -1215.194} C_VEL
LIN {X 0,Y 594.366,Z 43.449,A -85,B 0,C 180,E1 -1217.624,E2 -1217.624} C_VEL
LIN {X 0,Y 594.371,Z 43.442,A -85,B 0,C 180,E1 -1220.319,E2 -1220.319} C_VEL
LIN {X 0,Y 594.382,Z 43.445,A -85,B 0,C 180,E1 -1222.913,E2 -1222.913} C_VEL
LIN {X 0,Y 594.382,Z 43.441,A -85,B 0,C 180,E1 -1225.861,E2 -1225.861} C_VEL
LIN {X 0,Y 594.388,Z 43.443,A -85,B 0,C 180,E1 -1228.651,E2 -1228.651} C_VEL
LIN {X 0,Y 594.381,Z 43.45,A -85,B 0,C 180,E1 -1231.043,E2 -1231.043} C_VEL
LIN {X 0,Y 594.387,Z 43.44,A -85,B 0,C 180,E1 -1233.977,E2 -1233.977} C_VEL
LIN {X 0,Y 594.373,Z 43.444,A -85,B 0,C 180,E1 -1236.295,E2 -1236.295} C_VEL
LIN {X 0,Y 594.391,Z 43.442,A -85,B 0,C 180,E1 -1239.224,E2 -1239.224} C_VEL
LIN {X 0,Y 594.354,Z 43.446,A -85,B 0,C 180,E1 -1242.095,E2 -1242.095} C_VEL
LIN {X 0,Y 594.364,Z 43.447,A -85,B 0,C 180,E1 -1244.219,E2 -1244.219} C_VEL
LIN {X 0,Y 594.378,Z 43.448,A -85,B 0,C 180,E1 -1246.321,E2 -1246.321} C_VEL
LIN {X 0,Y 594.363,Z 43.444,A -85,B 0,C 180,E1 -1249.095,E2 -1249.095} C_VEL
LIN {X 0,Y 594.412,Z 43.439,A -85,B 0,C 180,E1 -1251.843,E2 -1251.843} C_VEL
LIN {X 0,Y 594.378,Z 43.446,A -85,B 0,C 180,E1 -1254.572,E2 -1254.572} C_VEL
LIN {X 0,Y 594.402,Z 43.438,A -85,B 0,C 180,E1 -1257.289,E2 -1257.289} C_VEL
LIN {X 0,Y 594.417,Z 43.445,A -85,B 0,C 180,E1 -1260,E2 -1260} C_VEL
LIN {X 0,Y 594.389,Z 43.441,A -85,B 0,C 180,E1 -1262.711,E2 -1262.711} C_VEL
LIN {X 0,Y 594.395,Z 43.442,A -85,B 0,C 180,E1 -1265.428,E2 -1265.428} C_VEL
LIN {X 0,Y 594.379,Z 43.446,A -85,B 0,C 180,E1 -1268.157,E2 -1268.157} C_VEL
LIN {X 0,Y 594.379,Z 43.442,A -85,B 0,C 180,E1 -1271.068,E2 -1271.068} C_VEL
LIN {X 0,Y 594.372,Z 43.452,A -85,B 0,C 180,E1 -1273.679,E2 -1273.679} C_VEL
LIN {X 0,Y 594.346,Z 43.447,A -85,B 0,C 180,E1 -1275.299,E2 -1275.299} C_VEL
LIN {X 0,Y 593.676,Z 43.535,A -85,B 0,C 180,E1 -1275.865,E2 -1275.865} C_VEL
LIN {X 0,Y 590.808,Z 43.891,A -85,B 0,C 180,E1 -1276.783,E2 -1276.783} C_VEL
LIN {X 0,Y 588.395,Z 44.196,A -85,B 0,C 180,E1 -1277.522,E2 -1277.522} C_VEL
LIN {X 0,Y 587.372,Z 44.316,A -85,B 0,C 180,E1 -1278.092,E2 -1278.092} C_VEL
LIN {X 0,Y 587.296,Z 44.324,A -85,B 0,C 180,E1 -1278.285,E2 -1278.285} C_VEL
LIN {X 0,Y 587.332,Z 44.323,A -85,B 0,C 180,E1 -1281.038,E2 -1281.038} C_VEL
LIN {X 0,Y 587.301,Z 44.324,A -85,B 0,C 180,E1 -1284.008,E2 -1284.008} C_VEL
LIN {X 0,Y 587.334,Z 44.319,A -85,B 0,C 180,E1 -1286.279,E2 -1286.279} C_VEL
LIN {X 0,Y 587.346,Z 44.327,A -85,B 0,C 180,E1 -1289.133,E2 -1289.133} C_VEL
LIN {X 0,Y 587.34,Z 44.318,A -85,B 0,C 180,E1 -1291.835,E2 -1291.835} C_VEL
LIN {X 0,Y 587.338,Z 44.319,A -85,B 0,C 180,E1 -1294.346,E2 -1294.346} C_VEL
LIN {X 0,Y 587.34,Z 44.319,A -85,B 0,C 180,E1 -1297.609,E2 -1297.609} C_VEL
LIN {X 0,Y 587.306,Z 44.324,A -85,B 0,C 180,E1 -1300.256,E2 -1300.256} C_VEL
LIN {X 0,Y 587.305,Z 44.326,A -85,B 0,C 180,E1 -1303.117,E2 -1303.117} C_VEL
LIN {X 0,Y 587.314,Z 44.323,A -85,B 0,C 180,E1 -1306.049,E2 -1306.049} C_VEL
LIN {X 0,Y 587.333,Z 44.323,A -85,B 0,C 180,E1 -1308.926,E2 -1308.926} C_VEL
LIN {X 0,Y 587.314,Z 44.321,A -85,B 0,C 180,E1 -1311.52,E2 -1311.52} C_VEL
LIN {X 0,Y 587.282,Z 44.33,A -85,B 0,C 180,E1 -1314.099,E2 -1314.099} C_VEL
LIN {X 0,Y 587.332,Z 44.324,A -85,B 0,C 180,E1 -1316.603,E2 -1316.603} C_VEL
LIN {X 0,Y 587.335,Z 44.319,A -85,B 0,C 180,E1 -1319.491,E2 -1319.491} C_VEL
LIN {X 0,Y 587.304,Z 44.332,A -85,B 0,C 180,E1 -1322.18,E2 -1322.18} C_VEL
LIN {X 0,Y 587.307,Z 44.325,A -85,B 0,C 180,E1 -1324.482,E2 -1324.482} C_VEL
LIN {X 0,Y 587.312,Z 44.321,A -85,B 0,C 180,E1 -1327.134,E2 -1327.134} C_VEL
LIN {X 0,Y 587.322,Z 44.327,A -85,B 0,C 180,E1 -1329.695,E2 -1329.695} C_VEL
LIN {X 0,Y 587.288,Z 44.334,A -85,B 0,C 180,E1 -1331.872,E2 -1331.872} C_VEL
LIN {X 0,Y 587.305,Z 44.328,A -85,B 0,C 180,E1 -1334.024,E2 -1334.024} C_VEL
LIN {X 0,Y 587.332,Z 44.323,A -85,B 0,C 180,E1 -1336.154,E2 -1336.154} C_VEL
LIN {X 0,Y 587.336,Z 44.38,A -85,B 0,C 180,E1 -1338.781,E2 -1338.781} C_VEL
LIN {X 0,Y 587.403,Z 56.753,A -85,B 0,C 180,E1 -1341.052,E2 -1341.052} C_VEL
LIN {X 0,Y 587.309,Z 70.89,A -85,B 0,C 180,E1 -1343.572,E2 -1343.572} C_VEL
LIN {X 0,Y 587.859,Z 76.455,A -85,B 0,C 180,E1 -1343.654,E2 -1343.654} C_VEL
LIN {X 0,Y 587.702,Z 176.836,A -85,B 0,C 180,E1 -1344.898,E2 -1344.898} C_VEL
LIN {X 0,Y 587.664,Z 189.964,A -85,B 0,C 180,E1 -1345.198,E2 -1345.198} C_VEL
LIN {X 0,Y 587.61,Z 202.561,A -85,B 0,C 180,E1 -1345.627,E2 -1345.627} C_VEL
LIN {X 0,Y 587.571,Z 213.799,A -85,B 0,C 180,E1 -1346.142,E2 -1346.142} C_VEL
LIN {X 0,Y 587.475,Z 225.413,A -85,B 0,C 180,E1 -1346.828,E2 -1346.828} C_VEL
LIN {X 0,Y 587.374,Z 235.838,A -85,B 0,C 180,E1 -1347.6,E2 -1347.6} C_VEL
LIN {X 0,Y 587.315,Z 245.265,A -85,B 0,C 180,E1 -1348.457,E2 -1348.457} C_VEL
LIN {X 0,Y 587.259,Z 254.376,A -85,B 0,C 180,E1 -1349.486,E2 -1349.486} C_VEL
LIN {X 0,Y 587.254,Z 261.724,A -85,B 0,C 180,E1 -1350.514,E2 -1350.514} C_VEL
LIN {X 0,Y 587.204,Z 268.52,A -85,B 0,C 180,E1 -1351.715,E2 -1351.715} C_VEL
LIN {X 0,Y 587.145,Z 273.02,A -85,B 0,C 180,E1 -1352.745,E2 -1352.745} C_VEL
LIN {X 0,Y 587.19,Z 275.394,A -85,B 0,C 180,E1 -1353.431,E2 -1353.431} C_VEL
LIN {X 0,Y 587.171,Z 277.343,A -85,B 0,C 180,E1 -1354.118,E2 -1354.118} C_VEL
LIN {X 0,Y 587.127,Z 278.881,A -85,B 0,C 180,E1 -1354.807,E2 -1354.807} C_VEL
LIN {X 0,Y 587.169,Z 279.979,A -85,B 0,C 180,E1 -1355.495,E2 -1355.495} C_VEL
LIN {X 0,Y 587.167,Z 280.968,A -85,B 0,C 180,E1 -1356.875,E2 -1356.875} C_VEL
LIN {X 0,Y 587.146,Z 280.885,A -85,B 0,C 180,E1 -1357.566,E2 -1357.566} C_VEL
LIN {X 0,Y 587.139,Z 280.365,A -85,B 0,C 180,E1 -1358.259,E2 -1358.259} C_VEL
LIN {X 0,Y 587.129,Z 279.444,A -85,B 0,C 180,E1 -1358.952,E2 -1358.952} C_VEL
LIN {X 0,Y 587.154,Z 278.118,A -85,B 0,C 180,E1 -1359.647,E2 -1359.647} C_VEL
LIN {X 0,Y 587.185,Z 275.292,A -85,B 0,C 180,E1 -1360.692,E2 -1360.692} C_VEL
LIN {X 0,Y 587.178,Z 271.407,A -85,B 0,C 180,E1 -1361.74,E2 -1361.74} C_VEL
LIN {X 0,Y 587.193,Z 266.348,A -85,B 0,C 180,E1 -1362.793,E2 -1362.793} C_VEL
LIN {X 0,Y 587.238,Z 259.95,A -85,B 0,C 180,E1 -1363.849,E2 -1363.849} C_VEL
LIN {X 0,Y 587.288,Z 251.87,A -85,B 0,C 180,E1 -1364.909,E2 -1364.909} C_VEL
LIN {X 0,Y 587.313,Z 243.576,A -85,B 0,C 180,E1 -1365.798,E2 -1365.798} C_VEL
LIN {X 0,Y 587.429,Z 233.407,A -85,B 0,C 180,E1 -1366.687,E2 -1366.687} C_VEL
LIN {X 0,Y 587.434,Z 223.255,A -85,B 0,C 180,E1 -1367.404,E2 -1367.404} C_VEL
LIN {X 0,Y 587.553,Z 212.164,A -85,B 0,C 180,E1 -1368.03,E2 -1368.03} C_VEL
LIN {X 0,Y 587.646,Z 199.837,A -85,B 0,C 180,E1 -1368.568,E2 -1368.568} C_VEL
LIN {X 0,Y 587.684,Z 186.837,A -85,B 0,C 180,E1 -1368.978,E2 -1368.978} C_VEL
LIN {X 0,Y 587.73,Z 173.436,A -85,B 0,C 180,E1 -1369.243,E2 -1369.243} C_VEL
LIN {X 0,Y 587.715,Z 72.997,A -85,B 0,C 180,E1 -1370.482,E2 -1370.482} C_VEL
LIN {X 0,Y 587.352,Z 70.586,A -85,B 0,C 180,E1 -1370.533,E2 -1370.533} C_VEL
LIN {X 0,Y 587.39,Z 55.558,A -85,B 0,C 180,E1 -1373.256,E2 -1373.256} C_VEL
LIN {X 0,Y 587.361,Z 44.795,A -85,B 0,C 180,E1 -1375.231,E2 -1375.231} C_VEL
LIN {X 0,Y 587.294,Z 44.328,A -85,B 0,C 180,E1 -1375.329,E2 -1375.329} C_VEL
LIN {X 0,Y 587.287,Z 44.328,A -85,B 0,C 180,E1 -1377.821,E2 -1377.821} C_VEL
LIN {X 0,Y 587.317,Z 44.328,A -85,B 0,C 180,E1 -1380.506,E2 -1380.506} C_VEL
LIN {X 0,Y 587.307,Z 44.323,A -85,B 0,C 180,E1 -1383.399,E2 -1383.399} C_VEL
LIN {X 0,Y 587.273,Z 44.333,A -85,B 0,C 180,E1 -1385.902,E2 -1385.902} C_VEL
LIN {X 0,Y 587.284,Z 44.328,A -85,B 0,C 180,E1 -1388.483,E2 -1388.483} C_VEL
LIN {X 0,Y 587.288,Z 44.325,A -85,B 0,C 180,E1 -1391.161,E2 -1391.161} C_VEL
LIN {X 0,Y 587.288,Z 44.328,A -85,B 0,C 180,E1 -1394.109,E2 -1394.109} C_VEL
LIN {X 0,Y 587.285,Z 44.326,A -85,B 0,C 180,E1 -1396.99,E2 -1396.99} C_VEL
LIN {X 0,Y 587.283,Z 44.329,A -85,B 0,C 180,E1 -1399.986,E2 -1399.986} C_VEL
LIN {X 0,Y 587.261,Z 44.328,A -85,B 0,C 180,E1 -1402.386,E2 -1402.386} C_VEL
LIN {X 0,Y 587.293,Z 44.326,A -85,B 0,C 180,E1 -1404.942,E2 -1404.942} C_VEL
LIN {X 0,Y 587.316,Z 44.329,A -85,B 0,C 180,E1 -1407.419,E2 -1407.419} C_VEL
LIN {X 0,Y 587.292,Z 44.326,A -85,B 0,C 180,E1 -1409.827,E2 -1409.827} C_VEL
LIN {X 0,Y 587.3,Z 44.323,A -85,B 0,C 180,E1 -1412.317,E2 -1412.317} C_VEL
LIN {X 0,Y 587.287,Z 44.331,A -85,B 0,C 180,E1 -1415.238,E2 -1415.238} C_VEL
LIN {X 0,Y 587.305,Z 44.324,A -85,B 0,C 180,E1 -1417.484,E2 -1417.484} C_VEL
LIN {X 0,Y 587.307,Z 44.322,A -85,B 0,C 180,E1 -1419.694,E2 -1419.694} C_VEL
LIN {X 0,Y 587.281,Z 44.325,A -85,B 0,C 180,E1 -1421.872,E2 -1421.872} C_VEL
LIN {X 0,Y 587.296,Z 44.324,A -85,B 0,C 180,E1 -1424.024,E2 -1424.024} C_VEL
LIN {X 0,Y 587.285,Z 44.33,A -85,B 0,C 180,E1 -1426.857,E2 -1426.857} C_VEL
LIN {X 0,Y 587.341,Z 44.321,A -85,B 0,C 180,E1 -1428.962,E2 -1428.962} C_VEL
LIN {X 0,Y 587.316,Z 44.322,A -85,B 0,C 180,E1 -1431.744,E2 -1431.744} C_VEL
LIN {X 0,Y 587.348,Z 44.324,A -85,B 0,C 180,E1 -1434.507,E2 -1434.507} C_VEL
LIN {X 0,Y 587.346,Z 44.317,A -85,B 0,C 180,E1 -1437.256,E2 -1437.256} C_VEL
LIN {X 0,Y 587.376,Z 44.32,A -85,B 0,C 180,E1 -1440,E2 -1440} C_VEL
LIN {X 0,Y 587.359,Z 44.317,A -85,B 0,C 180,E1 -1442.743,E2 -1442.743} C_VEL
LIN {X 0,Y 587.334,Z 44.321,A -85,B 0,C 180,E1 -1445.493,E2 -1445.493} C_VEL
LIN {X 0,Y 587.34,Z 44.322,A -85,B 0,C 180,E1 -1448.256,E2 -1448.256} C_VEL
LIN {X 0,Y 587.334,Z 44.319,A -85,B 0,C 180,E1 -1451.124,E2 -1451.124} C_VEL
LIN {X 0,Y 587.355,Z 44.323,A -85,B 0,C 180,E1 -1453.846,E2 -1453.846} C_VEL
LIN {X 0,Y 587.319,Z 44.32,A -85,B 0,C 180,E1 -1456.803,E2 -1456.803} C_VEL
LIN {X 0,Y 587.308,Z 44.33,A -85,B 0,C 180,E1 -1459.576,E2 -1459.576} C_VEL
LIN {X 0,Y 587.315,Z 44.324,A -85,B 0,C 180,E1 -1461.775,E2 -1461.775} C_VEL
LIN {X 0,Y 587.316,Z 44.323,A -85,B 0,C 180,E1 -1464.76,E2 -1464.76} C_VEL
LIN {X 0,Y 587.339,Z 44.319,A -85,B 0,C 180,E1 -1467.818,E2 -1467.818} C_VEL
LIN {X 0,Y 587.323,Z 44.322,A -85,B 0,C 180,E1 -1470.507,E2 -1470.507} C_VEL
LIN {X 0,Y 587.334,Z 44.322,A -85,B 0,C 180,E1 -1473.397,E2 -1473.397} C_VEL
LIN {X 0,Y 587.291,Z 44.322,A -85,B 0,C 180,E1 -1475.9,E2 -1475.9} C_VEL
LIN {X 0,Y 587.321,Z 44.324,A -85,B 0,C 180,E1 -1478.48,E2 -1478.48} C_VEL
LIN {X 0,Y 587.337,Z 44.321,A -85,B 0,C 180,E1 -1481.157,E2 -1481.157} C_VEL
LIN {X 0,Y 587.315,Z 44.324,A -85,B 0,C 180,E1 -1484.112,E2 -1484.112} C_VEL
LIN {X 0,Y 587.314,Z 44.324,A -85,B 0,C 180,E1 -1486.993,E2 -1486.993} C_VEL
LIN {X 0,Y 587.316,Z 44.322,A -85,B 0,C 180,E1 -1489.745,E2 -1489.745} C_VEL
LIN {X 0,Y 587.345,Z 44.326,A -85,B 0,C 180,E1 -1492.392,E2 -1492.392} C_VEL
LIN {X 0,Y 587.348,Z 44.319,A -85,B 0,C 180,E1 -1495.653,E2 -1495.653} C_VEL
LIN {X 0,Y 587.34,Z 44.327,A -85,B 0,C 180,E1 -1498.231,E2 -1498.231} C_VEL
LIN {X 0,Y 587.348,Z 44.318,A -85,B 0,C 180,E1 -1500.867,E2 -1500.867} C_VEL
LIN {X 0,Y 587.34,Z 44.325,A -85,B 0,C 180,E1 -1503.721,E2 -1503.721} C_VEL
LIN {X 0,Y 587.374,Z 44.462,A -85,B 0,C 180,E1 -1506.486,E2 -1506.486} C_VEL
LIN {X 0,Y 587.838,Z 48.166,A -85,B 0,C 180,E1 -1507.013,E2 -1507.013} C_VEL
LIN {X 0,Y 587.746,Z 68.072,A -85,B 0,C 180,E1 -1509.71,E2 -1509.71} C_VEL
LIN {X 0,Y 587.588,Z 89.352,A -85,B 0,C 180,E1 -1512.601,E2 -1512.601} C_VEL
LIN {X 0,Y 587.457,Z 107.966,A -85,B 0,C 180,E1 -1515.095,E2 -1515.095} C_VEL
LIN {X 0,Y 587.401,Z 118.437,A -85,B 0,C 180,E1 -1516.486,E2 -1516.486} C_VEL
LIN {X 0,Y 587.84,Z 122.7,A -85,B 0,C 180,E1 -1516.562,E2 -1516.562} C_VEL
LIN {X 0,Y 587.755,Z 226.934,A -85,B 0,C 180,E1 -1517.855,E2 -1517.855} C_VEL
LIN {X 0,Y 587.672,Z 240.211,A -85,B 0,C 180,E1 -1518.16,E2 -1518.16} C_VEL
LIN {X 0,Y 587.629,Z 252.628,A -85,B 0,C 180,E1 -1518.585,E2 -1518.585} C_VEL
LIN {X 0,Y 587.558,Z 264.624,A -85,B 0,C 180,E1 -1519.141,E2 -1519.141} C_VEL
LIN {X 0,Y 587.461,Z 276.199,A -85,B 0,C 180,E1 -1519.836,E2 -1519.836} C_VEL
LIN {X 0,Y 587.366,Z 286.597,A -85,B 0,C 180,E1 -1520.617,E2 -1520.617} C_VEL
LIN {X 0,Y 587.322,Z 295.11,A -85,B 0,C 180,E1 -1521.397,E2 -1521.397} C_VEL
LIN {X 0,Y 587.274,Z 302.959,A -85,B 0,C 180,E1 -1522.263,E2 -1522.263} C_VEL
LIN {X 0,Y 587.23,Z 309.467,A -85,B 0,C 180,E1 -1523.126,E2 -1523.126} C_VEL
LIN {X 0,Y 587.237,Z 315.866,A -85,B 0,C 180,E1 -1524.161,E2 -1524.161} C_VEL
LIN {X 0,Y 587.147,Z 320.949,A -85,B 0,C 180,E1 -1525.193,E2 -1525.193} C_VEL
LIN {X 0,Y 587.213,Z 324.895,A -85,B 0,C 180,E1 -1526.225,E2 -1526.225} C_VEL
LIN {X 0,Y 587.132,Z 327.808,A -85,B 0,C 180,E1 -1527.255,E2 -1527.255} C_VEL
LIN {X 0,Y 587.141,Z 329.199,A -85,B 0,C 180,E1 -1527.942,E2 -1527.942} C_VEL
LIN {X 0,Y 587.14,Z 330.785,A -85,B 0,C 180,E1 -1529.314,E2 -1529.314} C_VEL
LIN {X 0,Y 587.137,Z 331,A -85,B 0,C 180,E1 -1530,E2 -1530} C_VEL
LIN {X 0,Y 587.147,Z 330.186,A -85,B 0,C 180,E1 -1531.372,E2 -1531.372} C_VEL
LIN {X 0,Y 587.141,Z 329.2,A -85,B 0,C 180,E1 -1532.058,E2 -1532.058} C_VEL
LIN {X 0,Y 587.132,Z 327.81,A -85,B 0,C 180,E1 -1532.744,E2 -1532.744} C_VEL
LIN {X 0,Y 587.213,Z 324.896,A -85,B 0,C 180,E1 -1533.774,E2 -1533.774} C_VEL
LIN {X 0,Y 587.147,Z 320.95,A -85,B 0,C 180,E1 -1534.806,E2 -1534.806} C_VEL
LIN {X 0,Y 587.218,Z 314.878,A -85,B 0,C 180,E1 -1536.011,E2 -1536.011} C_VEL
LIN {X 0,Y 587.245,Z 308.239,A -85,B 0,C 180,E1 -1537.046,E2 -1537.046} C_VEL
LIN {X 0,Y 587.299,Z 299.992,A -85,B 0,C 180,E1 -1538.083,E2 -1538.083} C_VEL
LIN {X 0,Y 587.343,Z 291.54,A -85,B 0,C 180,E1 -1538.949,E2 -1538.949} C_VEL
LIN {X 0,Y 587.416,Z 281.1,A -85,B 0,C 180,E1 -1539.816,E2 -1539.816} C_VEL
LIN {X 0,Y 587.481,Z 270.758,A -85,B 0,C 180,E1 -1540.511,E2 -1540.511} C_VEL
LIN {X 0,Y 587.561,Z 258.819,A -85,B 0,C 180,E1 -1541.149,E2 -1541.149} C_VEL
LIN {X 0,Y 587.63,Z 246.603,A -85,B 0,C 180,E1 -1541.639,E2 -1541.639} C_VEL
LIN {X 0,Y 587.728,Z 233.442,A -85,B 0,C 180,E1 -1542.013,E2 -1542.013} C_VEL
LIN {X 0,Y 587.776,Z 221.098,A -85,B 0,C 180,E1 -1542.231,E2 -1542.231} C_VEL
LIN {X 0,Y 587.714,Z 120.721,A -85,B 0,C 180,E1 -1543.465,E2 -1543.465} C_VEL
LIN {X 0,Y 587.401,Z 118.44,A -85,B 0,C 180,E1 -1543.514,E2 -1543.514} C_VEL
LIN {X 0,Y 587.549,Z 96.003,A -85,B 0,C 180,E1 -1546.504,E2 -1546.504} C_VEL
LIN {X 0,Y 587.668,Z 76.571,A -85,B 0,C 180,E1 -1549.131,E2 -1549.131} C_VEL
LIN {X 0,Y 587.827,Z 55.86,A -85,B 0,C 180,E1 -1551.939,E2 -1551.939} C_VEL
LIN {X 0,Y 587.711,Z 46.362,A -85,B 0,C 180,E1 -1553.242,E2 -1553.242} C_VEL
LIN {X 0,Y 587.366,Z 44.322,A -85,B 0,C 180,E1 -1553.537,E2 -1553.537} C_VEL
LIN {X 0,Y 587.339,Z 44.326,A -85,B 0,C 180,E1 -1556.278,E2 -1556.278} C_VEL
LIN {X 0,Y 587.35,Z 44.317,A -85,B 0,C 180,E1 -1559.133,E2 -1559.133} C_VEL
LIN {X 0,Y 587.347,Z 44.325,A -85,B 0,C 180,E1 -1561.836,E2 -1561.836} C_VEL
LIN {X 0,Y 587.347,Z 44.319,A -85,B 0,C 180,E1 -1564.347,E2 -1564.347} C_VEL
LIN {X 0,Y 587.345,Z 44.325,A -85,B 0,C 180,E1 -1567.607,E2 -1567.607} C_VEL
LIN {X 0,Y 587.316,Z 44.322,A -85,B 0,C 180,E1 -1570.254,E2 -1570.254} C_VEL
LIN {X 0,Y 587.314,Z 44.324,A -85,B 0,C 180,E1 -1573.118,E2 -1573.118} C_VEL
LIN {X 0,Y 587.312,Z 44.323,A -85,B 0,C 180,E1 -1576.048,E2 -1576.048} C_VEL
LIN {X 0,Y 587.336,Z 44.321,A -85,B 0,C 180,E1 -1578.925,E2 -1578.925} C_VEL
LIN {X 0,Y 587.32,Z 44.327,A -85,B 0,C 180,E1 -1581.52,E2 -1581.52} C_VEL
LIN {X 0,Y 587.293,Z 44.324,A -85,B 0,C 180,E1 -1584.1,E2 -1584.1} C_VEL
LIN {X 0,Y 587.334,Z 44.321,A -85,B 0,C 180,E1 -1586.603,E2 -1586.603} C_VEL
LIN {X 0,Y 587.335,Z 44.328,A -85,B 0,C 180,E1 -1589.034,E2 -1589.034} C_VEL
LIN {X 0,Y 587.318,Z 44.324,A -85,B 0,C 180,E1 -1591.403,E2 -1591.403} C_VEL
LIN {X 0,Y 587.36,Z 44.315,A -85,B 0,C 180,E1 -1593.819,E2 -1593.819} C_VEL
LIN {X 0,Y 587.327,Z 44.32,A -85,B 0,C 180,E1 -1595.993,E2 -1595.993} C_VEL
LIN {X 0,Y 587.315,Z 44.323,A -85,B 0,C 180,E1 -1598.225,E2 -1598.225} C_VEL
LIN {X 0,Y 587.342,Z 44.32,A -85,B 0,C 180,E1 -1601.151,E2 -1601.151} C_VEL
LIN {X 0,Y 587.317,Z 44.322,A -85,B 0,C 180,E1 -1604.025,E2 -1604.025} C_VEL
LIN {X 0,Y 587.309,Z 44.326,A -85,B 0,C 180,E1 -1606.858,E2 -1606.858} C_VEL
LIN {X 0,Y 587.337,Z 44.319,A -85,B 0,C 180,E1 -1609.66,E2 -1609.66} C_VEL
LIN {X 0,Y 587.35,Z 44.325,A -85,B 0,C 180,E1 -1612.437,E2 -1612.437} C_VEL
LIN {X 0,Y 587.353,Z 44.316,A -85,B 0,C 180,E1 -1615.195,E2 -1615.195} C_VEL
LIN {X 0,Y 587.372,Z 44.32,A -85,B 0,C 180,E1 -1617.943,E2 -1617.943} C_VEL
LIN {X 0,Y 587.376,Z 44.315,A -85,B 0,C 180,E1 -1620.686,E2 -1620.686} C_VEL
LIN {X 0,Y 587.329,Z 44.321,A -85,B 0,C 180,E1 -1623.43,E2 -1623.43} C_VEL
LIN {X 0,Y 587.316,Z 44.326,A -85,B 0,C 180,E1 -1626.183,E2 -1626.183} C_VEL
LIN {X 0,Y 587.339,Z 44.321,A -85,B 0,C 180,E1 -1628.256,E2 -1628.256} C_VEL
LIN {X 0,Y 587.349,Z 44.318,A -85,B 0,C 180,E1 -1631.134,E2 -1631.134} C_VEL
LIN {X 0,Y 587.332,Z 44.32,A -85,B 0,C 180,E1 -1634.248,E2 -1634.248} C_VEL
LIN {X 0,Y 587.338,Z 44.326,A -85,B 0,C 180,E1 -1637.407,E2 -1637.407} C_VEL
LIN {X 0,Y 587.296,Z 44.324,A -85,B 0,C 180,E1 -1638.285,E2 -1638.285} C_VEL
LIN {X 0,Y 586.66,Z 44.404,A -85,B 0,C 180,E1 -1638.857,E2 -1638.857} C_VEL
LIN {X 0,Y 583.851,Z 44.757,A -85,B 0,C 180,E1 -1639.786,E2 -1639.786} C_VEL
LIN {X 0,Y 581.446,Z 45.055,A -85,B 0,C 180,E1 -1640.533,E2 -1640.533} C_VEL
LIN {X 0,Y 580.385,Z 45.189,A -85,B 0,C 180,E1 -1641.109,E2 -1641.109} C_VEL
LIN {X 0,Y 580.284,Z 45.205,A -85,B 0,C 180,E1 -1641.304,E2 -1641.304} C_VEL
LIN {X 0,Y 580.261,Z 45.206,A -85,B 0,C 180,E1 -1643.559,E2 -1643.559} C_VEL
LIN {X 0,Y 580.288,Z 45.196,A -85,B 0,C 180,E1 -1646.333,E2 -1646.333} C_VEL
LIN {X 0,Y 580.294,Z 45.203,A -85,B 0,C 180,E1 -1649.309,E2 -1649.309} C_VEL
LIN {X 0,Y 580.296,Z 45.195,A -85,B 0,C 180,E1 -1652.201,E2 -1652.201} C_VEL
LIN {X 0,Y 580.286,Z 45.201,A -85,B 0,C 180,E1 -1654.697,E2 -1654.697} C_VEL
LIN {X 0,Y 580.296,Z 45.2,A -85,B 0,C 180,E1 -1657.269,E2 -1657.269} C_VEL
LIN {X 0,Y 580.286,Z 45.199,A -85,B 0,C 180,E1 -1660.27,E2 -1660.27} C_VEL
LIN {X 0,Y 580.274,Z 45.208,A -85,B 0,C 180,E1 -1662.707,E2 -1662.707} C_VEL
LIN {X 0,Y 580.257,Z 45.2,A -85,B 0,C 180,E1 -1665.611,E2 -1665.611} C_VEL
LIN {X 0,Y 580.273,Z 45.206,A -85,B 0,C 180,E1 -1668.67,E2 -1668.67} C_VEL
LIN {X 0,Y 580.269,Z 45.201,A -85,B 0,C 180,E1 -1670.965,E2 -1670.965} C_VEL
LIN {X 0,Y 580.243,Z 45.202,A -85,B 0,C 180,E1 -1673.595,E2 -1673.595} C_VEL
LIN {X 0,Y 580.311,Z 45.2,A -85,B 0,C 180,E1 -1676.145,E2 -1676.145} C_VEL
LIN {X 0,Y 580.271,Z 45.202,A -85,B 0,C 180,E1 -1678.614,E2 -1678.614} C_VEL
LIN {X 0,Y 580.288,Z 45.196,A -85,B 0,C 180,E1 -1681.024,E2 -1681.024} C_VEL
LIN {X 0,Y 580.253,Z 45.209,A -85,B 0,C 180,E1 -1684.149,E2 -1684.149} C_VEL
LIN {X 0,Y 580.269,Z 45.202,A -85,B 0,C 180,E1 -1686.442,E2 -1686.442} C_VEL
LIN {X 0,Y 580.272,Z 45.201,A -85,B 0,C 180,E1 -1689.437,E2 -1689.437} C_VEL
LIN {X 0,Y 580.249,Z 45.208,A -85,B 0,C 180,E1 -1691.645,E2 -1691.645} C_VEL
LIN {X 0,Y 580.282,Z 45.198,A -85,B 0,C 180,E1 -1694.547,E2 -1694.547} C_VEL
LIN {X 0,Y 580.294,Z 45.203,A -85,B 0,C 180,E1 -1697.409,E2 -1697.409} C_VEL
LIN {X 0,Y 580.314,Z 45.294,A -85,B 0,C 180,E1 -1698.708,E2 -1698.708} C_VEL
LIN {X 0,Y 580.345,Z 55.338,A -85,B 0,C 180,E1 -1700.591,E2 -1700.591} C_VEL
LIN {X 0,Y 580.251,Z 70.626,A -85,B 0,C 180,E1 -1703.396,E2 -1703.396} C_VEL
LIN {X 0,Y 580.931,Z 75.908,A -85,B 0,C 180,E1 -1703.484,E2 -1703.484} C_VEL
LIN {X 0,Y 580.775,Z 176.787,A -85,B 0,C 180,E1 -1704.749,E2 -1704.749} C_VEL
LIN {X 0,Y 580.731,Z 189.929,A -85,B 0,C 180,E1 -1705.054,E2 -1705.054} C_VEL
LIN {X 0,Y 580.652,Z 202.543,A -85,B 0,C 180,E1 -1705.488,E2 -1705.488} C_VEL
LIN {X 0,Y 580.602,Z 213.786,A -85,B 0,C 180,E1 -1706.009,E2 -1706.009} C_VEL
LIN {X 0,Y 580.48,Z 225.401,A -85,B 0,C 180,E1 -1706.703,E2 -1706.703} C_VEL
LIN {X 0,Y 580.353,Z 235.833,A -85,B 0,C 180,E1 -1707.484,E2 -1707.484} C_VEL
LIN {X 0,Y 580.263,Z 246.101,A -85,B 0,C 180,E1 -1708.439,E2 -1708.439} C_VEL
LIN {X 0,Y 580.196,Z 255.045,A -85,B 0,C 180,E1 -1709.48,E2 -1709.48} C_VEL
LIN {X 0,Y 580.188,Z 262.274,A -85,B 0,C 180,E1 -1710.521,E2 -1710.521} C_VEL
LIN {X 0,Y 580.107,Z 268.921,A -85,B 0,C 180,E1 -1711.736,E2 -1711.736} C_VEL
LIN {X 0,Y 580.056,Z 273.328,A -85,B 0,C 180,E1 -1712.778,E2 -1712.778} C_VEL
LIN {X 0,Y 580.115,Z 275.657,A -85,B 0,C 180,E1 -1713.473,E2 -1713.473} C_VEL
LIN {X 0,Y 580.088,Z 277.563,A -85,B 0,C 180,E1 -1714.169,E2 -1714.169} C_VEL
LIN {X 0,Y 580.03,Z 279.043,A -85,B 0,C 180,E1 -1714.866,E2 -1714.866} C_VEL
LIN {X 0,Y 580.09,Z 280.077,A -85,B 0,C 180,E1 -1715.562,E2 -1715.562} C_VEL
LIN {X 0,Y 580.061,Z 280.987,A -85,B 0,C 180,E1 -1716.959,E2 -1716.959} C_VEL
LIN {X 0,Y 580.067,Z 280.839,A -85,B 0,C 180,E1 -1717.659,E2 -1717.659} C_VEL
LIN {X 0,Y 580.061,Z 280.268,A -85,B 0,C 180,E1 -1718.36,E2 -1718.36} C_VEL
LIN {X 0,Y 580.064,Z 277.935,A -85,B 0,C 180,E1 -1719.766,E2 -1719.766} C_VEL
LIN {X 0,Y 580.071,Z 274.18,A -85,B 0,C 180,E1 -1721.072,E2 -1721.072} C_VEL
LIN {X 0,Y 580.109,Z 269.447,A -85,B 0,C 180,E1 -1722.241,E2 -1722.241} C_VEL
LIN {X 0,Y 580.132,Z 263.85,A -85,B 0,C 180,E1 -1723.308,E2 -1723.308} C_VEL
LIN {X 0,Y 580.216,Z 256.236,A -85,B 0,C 180,E1 -1724.456,E2 -1724.456} C_VEL
LIN {X 0,Y 580.251,Z 247.931,A -85,B 0,C 180,E1 -1725.454,E2 -1725.454} C_VEL
LIN {X 0,Y 580.333,Z 237.763,A -85,B 0,C 180,E1 -1726.444,E2 -1726.444} C_VEL
LIN {X 0,Y 580.402,Z 227.832,A -85,B 0,C 180,E1 -1727.221,E2 -1727.221} C_VEL
LIN {X 0,Y 580.521,Z 217.247,A -85,B 0,C 180,E1 -1727.891,E2 -1727.891} C_VEL
LIN {X 0,Y 580.641,Z 205.433,A -85,B 0,C 180,E1 -1728.48,E2 -1728.48} C_VEL
LIN {X 0,Y 580.706,Z 193.36,A -85,B 0,C 180,E1 -1728.935,E2 -1728.935} C_VEL
LIN {X 0,Y 580.801,Z 180.792,A -85,B 0,C 180,E1 -1729.262,E2 -1729.262} C_VEL
LIN {X 0,Y 580.813,Z 164.771,A -85,B 0,C 180,E1 -1729.504,E2 -1729.504} C_VEL
LIN {X 0,Y 580.861,Z 74.028,A -85,B 0,C 180,E1 -1730.631,E2 -1730.631} C_VEL
LIN {X 0,Y 580.31,Z 70.607,A -85,B 0,C 180,E1 -1730.696,E2 -1730.696} C_VEL
LIN {X 0,Y 580.358,Z 55.035,A -85,B 0,C 180,E1 -1733.555,E2 -1733.555} C_VEL
LIN {X 0,Y 580.348,Z 45.872,A -85,B 0,C 180,E1 -1735.27,E2 -1735.27} C_VEL
LIN {X 0,Y 580.27,Z 45.203,A -85,B 0,C 180,E1 -1735.417,E2 -1735.417} C_VEL
LIN {X 0,Y 580.23,Z 45.212,A -85,B 0,C 180,E1 -1738.189,E2 -1738.189} C_VEL
LIN {X 0,Y 580.261,Z 45.204,A -85,B 0,C 180,E1 -1740.69,E2 -1740.69} C_VEL
LIN {X 0,Y 580.254,Z 45.202,A -85,B 0,C 180,E1 -1743.308,E2 -1743.308} C_VEL
LIN {X 0,Y 580.221,Z 45.209,A -85,B 0,C 180,E1 -1745.752,E2 -1745.752} C_VEL
LIN {X 0,Y 580.268,Z 45.207,A -85,B 0,C 180,E1 -1748.148,E2 -1748.148} C_VEL
LIN {X 0,Y 580.238,Z 45.203,A -85,B 0,C 180,E1 -1750.849,E2 -1750.849} C_VEL
LIN {X 0,Y 580.226,Z 45.212,A -85,B 0,C 180,E1 -1753.663,E2 -1753.663} C_VEL
LIN {X 0,Y 580.236,Z 45.205,A -85,B 0,C 180,E1 -1756.338,E2 -1756.338} C_VEL
LIN {X 0,Y 580.23,Z 45.206,A -85,B 0,C 180,E1 -1759.15,E2 -1759.15} C_VEL
LIN {X 0,Y 580.212,Z 45.211,A -85,B 0,C 180,E1 -1761.847,E2 -1761.847} C_VEL
LIN {X 0,Y 580.22,Z 45.205,A -85,B 0,C 180,E1 -1764.45,E2 -1764.45} C_VEL
LIN {X 0,Y 580.24,Z 45.206,A -85,B 0,C 180,E1 -1766.972,E2 -1766.972} C_VEL
LIN {X 0,Y 580.252,Z 45.208,A -85,B 0,C 180,E1 -1769.422,E2 -1769.422} C_VEL
LIN {X 0,Y 580.247,Z 45.201,A -85,B 0,C 180,E1 -1772.152,E2 -1772.152} C_VEL
LIN {X 0,Y 580.233,Z 45.21,A -85,B 0,C 180,E1 -1774.917,E2 -1774.917} C_VEL
LIN {X 0,Y 580.28,Z 45.203,A -85,B 0,C 180,E1 -1777.197,E2 -1777.197} C_VEL
LIN {X 0,Y 580.262,Z 45.202,A -85,B 0,C 180,E1 -1779.436,E2 -1779.436} C_VEL
LIN {X 0,Y 580.244,Z 45.202,A -85,B 0,C 180,E1 -1781.644,E2 -1781.644} C_VEL
LIN {X 0,Y 580.249,Z 45.201,A -85,B 0,C 180,E1 -1783.824,E2 -1783.824} C_VEL
LIN {X 0,Y 580.284,Z 45.198,A -85,B 0,C 180,E1 -1785.982,E2 -1785.982} C_VEL
LIN {X 0,Y 580.31,Z 45.199,A -85,B 0,C 180,E1 -1788.827,E2 -1788.827} C_VEL
LIN {X 0,Y 580.29,Z 45.196,A -85,B 0,C 180,E1 -1791.643,E2 -1791.643} C_VEL
LIN {X 0,Y 580.312,Z 45.202,A -85,B 0,C 180,E1 -1794.44,E2 -1794.44} C_VEL
LIN {X 0,Y 580.316,Z 45.193,A -85,B 0,C 180,E1 -1797.223,E2 -1797.223} C_VEL
LIN {X 0,Y 580.346,Z 45.195,A -85,B 0,C 180,E1 -1800,E2 -1800} C_VEL
LIN {X 0,Y 580.324,Z 45.193,A -85,B 0,C 180,E1 -1802.776,E2 -1802.776} C_VEL
LIN {X 0,Y 580.303,Z 45.197,A -85,B 0,C 180,E1 -1805.56,E2 -1805.56} C_VEL
LIN {X 0,Y 580.308,Z 45.197,A -85,B 0,C 180,E1 -1808.356,E2 -1808.356} C_VEL
LIN {X 0,Y 580.305,Z 45.195,A -85,B 0,C 180,E1 -1811.191,E2 -1811.191} C_VEL
LIN {X 0,Y 580.315,Z 45.198,A -85,B 0,C 180,E1 -1814.017,E2 -1814.017} C_VEL
LIN {X 0,Y 580.27,Z 45.199,A -85,B 0,C 180,E1 -1816.899,E2 -1816.899} C_VEL
LIN {X 0,Y 580.282,Z 45.201,A -85,B 0,C 180,E1 -1819.823,E2 -1819.823} C_VEL
LIN {X 0,Y 580.257,Z 45.2,A -85,B 0,C 180,E1 -1822.053,E2 -1822.053} C_VEL
LIN {X 0,Y 580.291,Z 45.203,A -85,B 0,C 180,E1 -1825.08,E2 -1825.08} C_VEL
LIN {X 0,Y 580.293,Z 45.196,A -85,B 0,C 180,E1 -1828.186,E2 -1828.186} C_VEL
LIN {X 0,Y 580.274,Z 45.202,A -85,B 0,C 180,E1 -1830.692,E2 -1830.692} C_VEL
LIN {X 0,Y 580.304,Z 45.199,A -85,B 0,C 180,E1 -1833.316,E2 -1833.316} C_VEL
LIN {X 0,Y 580.247,Z 45.2,A -85,B 0,C 180,E1 -1835.756,E2 -1835.756} C_VEL
LIN {X 0,Y 580.286,Z 45.197,A -85,B 0,C 180,E1 -1838.147,E2 -1838.147} C_VEL
LIN {X 0,Y 580.299,Z 45.203,A -85,B 0,C 180,E1 -1840.844,E2 -1840.844} C_VEL
LIN {X 0,Y 580.275,Z 45.198,A -85,B 0,C 180,E1 -1843.658,E2 -1843.658} C_VEL
LIN {X 0,Y 580.276,Z 45.206,A -85,B 0,C 180,E1 -1846.61,E2 -1846.61} C_VEL
LIN {X 0,Y 580.3,Z 45.196,A -85,B 0,C 180,E1 -1849.156,E2 -1849.156} C_VEL
LIN {X 0,Y 580.29,Z 45.2,A -85,B 0,C 180,E1 -1851.927,E2 -1851.927} C_VEL
LIN {X 0,Y 580.255,Z 45.207,A -85,B 0,C 180,E1 -1854.453,E2 -1854.453} C_VEL
LIN {X 0,Y 580.291,Z 45.197,A -85,B 0,C 180,E1 -1856.975,E2 -1856.975} C_VEL
LIN {X 0,Y 580.298,Z 45.198,A -85,B 0,C 180,E1 -1859.425,E2 -1859.425} C_VEL
LIN {X 0,Y 580.299,Z 45.203,A -85,B 0,C 180,E1 -1862.142,E2 -1862.142} C_VEL
LIN {X 0,Y 580.325,Z 45.195,A -85,B 0,C 180,E1 -1865.27,E2 -1865.27} C_VEL
LIN {X 0,Y 580.349,Z 45.349,A -85,B 0,C 180,E1 -1866.35,E2 -1866.35} C_VEL
LIN {X 0,Y 580.896,Z 49.642,A -85,B 0,C 180,E1 -1866.968,E2 -1866.968} C_VEL
LIN {X 0,Y 580.766,Z 67.762,A -85,B 0,C 180,E1 -1869.455,E2 -1869.455} C_VEL
LIN {X 0,Y 580.624,Z 89.352,A -85,B 0,C 180,E1 -1872.386,E2 -1872.386} C_VEL
LIN {X 0,Y 580.433,Z 109.296,A -85,B 0,C 180,E1 -1875.09,E2 -1875.09} C_VEL
LIN {X 0,Y 580.403,Z 118.52,A -85,B 0,C 180,E1 -1876.331,E2 -1876.331} C_VEL
LIN {X 0,Y 580.964,Z 124.489,A -85,B 0,C 180,E1 -1876.422,E2 -1876.422} C_VEL
LIN {X 0,Y 580.816,Z 226.934,A -85,B 0,C 180,E1 -1877.708,E2 -1877.708} C_VEL
LIN {X 0,Y 580.748,Z 240.21,A -85,B 0,C 180,E1 -1878.017,E2 -1878.017} C_VEL
LIN {X 0,Y 580.663,Z 251.911,A -85,B 0,C 180,E1 -1878.418,E2 -1878.418} C_VEL
LIN {X 0,Y 580.568,Z 262.928,A -85,B 0,C 180,E1 -1878.92,E2 -1878.92} C_VEL
LIN {X 0,Y 580.47,Z 273.583,A -85,B 0,C 180,E1 -1879.536,E2 -1879.536} C_VEL
LIN {X 0,Y 580.378,Z 284.468,A -85,B 0,C 180,E1 -1880.327,E2 -1880.327} C_VEL
LIN {X 0,Y 580.271,Z 295.11,A -85,B 0,C 180,E1 -1881.292,E2 -1881.292} C_VEL
LIN {X 0,Y 580.222,Z 302.959,A -85,B 0,C 180,E1 -1882.168,E2 -1882.168} C_VEL
LIN {X 0,Y 580.154,Z 310.65,A -85,B 0,C 180,E1 -1883.221,E2 -1883.221} C_VEL
LIN {X 0,Y 580.139,Z 317.679,A -85,B 0,C 180,E1 -1884.438,E2 -1884.438} C_VEL
LIN {X 0,Y 580.108,Z 322.371,A -85,B 0,C 180,E1 -1885.483,E2 -1885.483} C_VEL
LIN {X 0,Y 580.123,Z 325.957,A -85,B 0,C 180,E1 -1886.527,E2 -1886.527} C_VEL
LIN {X 0,Y 580.043,Z 327.808,A -85,B 0,C 180,E1 -1887.222,E2 -1887.222} C_VEL
LIN {X 0,Y 580.04,Z 329.197,A -85,B 0,C 180,E1 -1887.917,E2 -1887.917} C_VEL
LIN {X 0,Y 580.04,Z 330.785,A -85,B 0,C 180,E1 -1889.306,E2 -1889.306} C_VEL
LIN {X 0,Y 580.037,Z 331,A -85,B 0,C 180,E1 -1890,E2 -1890} C_VEL
LIN {X 0,Y 580.047,Z 330.186,A -85,B 0,C 180,E1 -1891.388,E2 -1891.388} C_VEL
LIN {X 0,Y 580.04,Z 329.199,A -85,B 0,C 180,E1 -1892.083,E2 -1892.083} C_VEL
LIN {X 0,Y 580.043,Z 327.81,A -85,B 0,C 180,E1 -1892.778,E2 -1892.778} C_VEL
LIN {X 0,Y 580.11,Z 324.896,A -85,B 0,C 180,E1 -1893.82,E2 -1893.82} C_VEL
LIN {X 0,Y 580.053,Z 320.95,A -85,B 0,C 180,E1 -1894.865,E2 -1894.865} C_VEL
LIN {X 0,Y 580.139,Z 314.878,A -85,B 0,C 180,E1 -1896.085,E2 -1896.085} C_VEL
LIN {X 0,Y 580.184,Z 308.239,A -85,B 0,C 180,E1 -1897.132,E2 -1897.132} C_VEL
LIN {X 0,Y 580.25,Z 299.992,A -85,B 0,C 180,E1 -1898.182,E2 -1898.182} C_VEL
LIN {X 0,Y 580.308,Z 291.541,A -85,B 0,C 180,E1 -1899.058,E2 -1899.058} C_VEL
LIN {X 0,Y 580.419,Z 281.099,A -85,B 0,C 180,E1 -1899.936,E2 -1899.936} C_VEL
LIN {X 0,Y 580.501,Z 270.756,A -85,B 0,C 180,E1 -1900.639,E2 -1900.639} C_VEL
LIN {X 0,Y 580.596,Z 259.248,A -85,B 0,C 180,E1 -1901.264,E2 -1901.264} C_VEL
LIN {X 0,Y 580.682,Z 246.477,A -85,B 0,C 180,E1 -1901.785,E2 -1901.785} C_VEL
LIN {X 0,Y 580.783,Z 233.44,A -85,B 0,C 180,E1 -1902.159,E2 -1902.159} C_VEL
LIN {X 0,Y 580.838,Z 221.098,A -85,B 0,C 180,E1 -1902.38,E2 -1902.38} C_VEL
LIN {X 0,Y 580.8,Z 121.394,A -85,B 0,C 180,E1 -1903.62,E2 -1903.62} C_VEL
LIN {X 0,Y 580.41,Z 118.44,A -85,B 0,C 180,E1 -1903.68,E2 -1903.68} C_VEL
LIN {X 0,Y 580.572,Z 96.003,A -85,B 0,C 180,E1 -1906.708,E2 -1906.708} C_VEL
LIN {X 0,Y 580.69,Z 77.223,A -85,B 0,C 180,E1 -1909.261,E2 -1909.261} C_VEL
LIN {X 0,Y 580.883,Z 56.911,A -85,B 0,C 180,E1 -1912.028,E2 -1912.028} C_VEL
LIN {X 0,Y 580.786,Z 47.87,A -85,B 0,C 180,E1 -1913.287,E2 -1913.287} C_VEL
LIN {X 0,Y 580.307,Z 45.202,A -85,B 0,C 180,E1 -1913.699,E2 -1913.699} C_VEL
LIN {X 0,Y 580.292,Z 45.203,A -85,B 0,C 180,E1 -1916.334,E2 -1916.334} C_VEL
LIN {X 0,Y 580.302,Z 45.196,A -85,B 0,C 180,E1 -1919.309,E2 -1919.309} C_VEL
LIN {X 0,Y 580.299,Z 45.2,A -85,B 0,C 180,E1 -1922.2,E2 -1922.2} C_VEL
LIN {X 0,Y 580.29,Z 45.196,A -85,B 0,C 180,E1 -1924.696,E2 -1924.696} C_VEL
LIN {X 0,Y 580.299,Z 45.198,A -85,B 0,C 180,E1 -1927.268,E2 -1927.268} C_VEL
LIN {X 0,Y 580.295,Z 45.197,A -85,B 0,C 180,E1 -1930.271,E2 -1930.271} C_VEL
LIN {X 0,Y 580.277,Z 45.198,A -85,B 0,C 180,E1 -1932.706,E2 -1932.706} C_VEL
LIN {X 0,Y 580.255,Z 45.208,A -85,B 0,C 180,E1 -1935.61,E2 -1935.61} C_VEL
LIN {X 0,Y 580.279,Z 45.198,A -85,B 0,C 180,E1 -1938.231,E2 -1938.231} C_VEL
LIN {X 0,Y 580.273,Z 45.202,A -85,B 0,C 180,E1 -1940.965,E2 -1940.965} C_VEL
LIN {X 0,Y 580.268,Z 45.203,A -85,B 0,C 180,E1 -1943.596,E2 -1943.596} C_VEL
LIN {X 0,Y 580.308,Z 45.194,A -85,B 0,C 180,E1 -1946.145,E2 -1946.145} C_VEL
LIN {X 0,Y 580.283,Z 45.2,A -85,B 0,C 180,E1 -1948.615,E2 -1948.615} C_VEL
LIN {X 0,Y 580.29,Z 45.206,A -85,B 0,C 180,E1 -1951.024,E2 -1951.024} C_VEL
LIN {X 0,Y 580.292,Z 45.196,A -85,B 0,C 180,E1 -1953.666,E2 -1953.666} C_VEL
LIN {X 0,Y 580.297,Z 45.195,A -85,B 0,C 180,E1 -1955.684,E2 -1955.684} C_VEL
LIN {X 0,Y 580.267,Z 45.199,A -85,B 0,C 180,E1 -1957.947,E2 -1957.947} C_VEL
LIN {X 0,Y 580.293,Z 45.202,A -85,B 0,C 180,E1 -1960.913,E2 -1960.913} C_VEL
LIN {X 0,Y 580.266,Z 45.199,A -85,B 0,C 180,E1 -1963.825,E2 -1963.825} C_VEL
LIN {X 0,Y 580.268,Z 45.206,A -85,B 0,C 180,E1 -1966.696,E2 -1966.696} C_VEL
LIN {X 0,Y 580.296,Z 45.195,A -85,B 0,C 180,E1 -1969.533,E2 -1969.533} C_VEL
LIN {X 0,Y 580.317,Z 45.203,A -85,B 0,C 180,E1 -1972.345,E2 -1972.345} C_VEL
LIN {X 0,Y 580.325,Z 45.192,A -85,B 0,C 180,E1 -1975.137,E2 -1975.137} C_VEL
LIN {X 0,Y 580.342,Z 45.196,A -85,B 0,C 180,E1 -1977.918,E2 -1977.918} C_VEL
LIN {X 0,Y 580.348,Z 45.19,A -85,B 0,C 180,E1 -1980.694,E2 -1980.694} C_VEL
LIN {X 0,Y 580.281,Z 45.2,A -85,B 0,C 180,E1 -1983.472,E2 -1983.472} C_VEL
LIN {X 0,Y 580.324,Z 45.196,A -85,B 0,C 180,E1 -1985.56,E2 -1985.56} C_VEL
LIN {X 0,Y 580.308,Z 45.196,A -85,B 0,C 180,E1 -1988.357,E2 -1988.357} C_VEL
LIN {X 0,Y 580.301,Z 45.197,A -85,B 0,C 180,E1 -1991.191,E2 -1991.191} C_VEL
LIN {X 0,Y 580.307,Z 45.198,A -85,B 0,C 180,E1 -1994.018,E2 -1994.018} C_VEL
LIN {X 0,Y 580.29,Z 45.197,A -85,B 0,C 180,E1 -1996.906,E2 -1996.906} C_VEL
LIN {X 0,Y 580.282,Z 45.201,A -85,B 0,C 180,E1 -1999.823,E2 -1999.823} C_VEL
LIN {X 0,Y 580.284,Z 45.205,A -85,B 0,C 180,E1 -2001.304,E2 -2001.304} C_VEL
LIN {X 0,Y 579.574,Z 45.3,A -85,B 0,C 180,E1 -2001.883,E2 -2001.883} C_VEL
LIN {X 0,Y 576.69,Z 45.656,A -85,B 0,C 180,E1 -2002.823,E2 -2002.823} C_VEL
LIN {X 0,Y 574.289,Z 45.95,A -85,B 0,C 180,E1 -2003.579,E2 -2003.579} C_VEL
LIN {X 0,Y 573.276,Z 46.07,A -85,B 0,C 180,E1 -2004.163,E2 -2004.163} C_VEL
LIN {X 0,Y 573.201,Z 46.079,A -85,B 0,C 180,E1 -2004.361,E2 -2004.361} C_VEL
LIN {X 0,Y 573.247,Z 46.079,A -85,B 0,C 180,E1 -2006.976,E2 -2006.976} C_VEL
LIN {X 0,Y 573.238,Z 46.079,A -85,B 0,C 180,E1 -2009.487,E2 -2009.487} C_VEL
LIN {X 0,Y 573.252,Z 46.076,A -85,B 0,C 180,E1 -2012.646,E2 -2012.646} C_VEL
LIN {X 0,Y 573.205,Z 46.085,A -85,B 0,C 180,E1 -2015.188,E2 -2015.188} C_VEL
LIN {X 0,Y 573.232,Z 46.075,A -85,B 0,C 180,E1 -2017.808,E2 -2017.808} C_VEL
LIN {X 0,Y 573.247,Z 46.079,A -85,B 0,C 180,E1 -2020.525,E2 -2020.525} C_VEL
LIN {X 0,Y 573.21,Z 46.079,A -85,B 0,C 180,E1 -2023.362,E2 -2023.362} C_VEL
LIN {X 0,Y 573.236,Z 46.08,A -85,B 0,C 180,E1 -2026.333,E2 -2026.333} C_VEL
LIN {X 0,Y 573.247,Z 46.073,A -85,B 0,C 180,E1 -2029.475,E2 -2029.475} C_VEL
LIN {X 0,Y 573.222,Z 46.082,A -85,B 0,C 180,E1 -2032.192,E2 -2032.192} C_VEL
LIN {X 0,Y 573.226,Z 46.076,A -85,B 0,C 180,E1 -2035.231,E2 -2035.231} C_VEL
LIN {X 0,Y 573.249,Z 46.076,A -85,B 0,C 180,E1 -2037.773,E2 -2037.773} C_VEL
LIN {X 0,Y 573.262,Z 46.075,A -85,B 0,C 180,E1 -2040.634,E2 -2040.634} C_VEL
LIN {X 0,Y 573.201,Z 46.081,A -85,B 0,C 180,E1 -2043.516,E2 -2043.516} C_VEL
LIN {X 0,Y 573.225,Z 46.084,A -85,B 0,C 180,E1 -2046.134,E2 -2046.134} C_VEL
LIN {X 0,Y 573.252,Z 46.073,A -85,B 0,C 180,E1 -2049.174,E2 -2049.174} C_VEL
LIN {X 0,Y 573.208,Z 46.082,A -85,B 0,C 180,E1 -2051.411,E2 -2051.411} C_VEL
LIN {X 0,Y 573.222,Z 46.079,A -85,B 0,C 180,E1 -2054.352,E2 -2054.352} C_VEL
LIN {X 0,Y 573.21,Z 46.08,A -85,B 0,C 180,E1 -2056.529,E2 -2056.529} C_VEL
LIN {X 0,Y 573.273,Z 46.171,A -85,B 0,C 180,E1 -2058.621,E2 -2058.621} C_VEL
LIN {X 0,Y 573.416,Z 52.187,A -85,B 0,C 180,E1 -2059.763,E2 -2059.763} C_VEL
LIN {X 0,Y 573.269,Z 67.284,A -85,B 0,C 180,E1 -2062.604,E2 -2062.604} C_VEL
LIN {X 0,Y 573.263,Z 70.913,A -85,B 0,C 180,E1 -2063.236,E2 -2063.236} C_VEL
LIN {X 0,Y 574.057,Z 77.049,A -85,B 0,C 180,E1 -2063.333,E2 -2063.333} C_VEL
LIN {X 0,Y 573.843,Z 176.743,A -85,B 0,C 180,E1 -2064.598,E2 -2064.598} C_VEL
LIN {X 0,Y 573.76,Z 189.913,A -85,B 0,C 180,E1 -2064.905,E2 -2064.905} C_VEL
LIN {X 0,Y 573.694,Z 202.526,A -85,B 0,C 180,E1 -2065.345,E2 -2065.345} C_VEL
LIN {X 0,Y 573.632,Z 213.774,A -85,B 0,C 180,E1 -2065.873,E2 -2065.873} C_VEL
LIN {X 0,Y 573.481,Z 225.39,A -85,B 0,C 180,E1 -2066.575,E2 -2066.575} C_VEL
LIN {X 0,Y 573.34,Z 235.824,A -85,B 0,C 180,E1 -2067.366,E2 -2067.366} C_VEL
LIN {X 0,Y 573.243,Z 245.255,A -85,B 0,C 180,E1 -2068.244,E2 -2068.244} C_VEL
LIN {X 0,Y 573.161,Z 254.368,A -85,B 0,C 180,E1 -2069.298,E2 -2069.298} C_VEL
LIN {X 0,Y 573.128,Z 261.715,A -85,B 0,C 180,E1 -2070.352,E2 -2070.352} C_VEL
LIN {X 0,Y 572.993,Z 267.638,A -85,B 0,C 180,E1 -2071.406,E2 -2071.406} C_VEL
LIN {X 0,Y 573.028,Z 272.323,A -85,B 0,C 180,E1 -2072.46,E2 -2072.46} C_VEL
LIN {X 0,Y 573.014,Z 275.921,A -85,B 0,C 180,E1 -2073.516,E2 -2073.516} C_VEL
LIN {X 0,Y 573.008,Z 277.781,A -85,B 0,C 180,E1 -2074.22,E2 -2074.22} C_VEL
LIN {X 0,Y 572.938,Z 279.182,A -85,B 0,C 180,E1 -2074.926,E2 -2074.926} C_VEL
LIN {X 0,Y 572.992,Z 280.176,A -85,B 0,C 180,E1 -2075.631,E2 -2075.631} C_VEL
LIN {X 0,Y 572.972,Z 281,A -85,B 0,C 180,E1 -2077.046,E2 -2077.046} C_VEL
LIN {X 0,Y 572.978,Z 280.781,A -85,B 0,C 180,E1 -2077.754,E2 -2077.754} C_VEL
LIN {X 0,Y 572.929,Z 279.16,A -85,B 0,C 180,E1 -2079.176,E2 -2079.176} C_VEL
LIN {X 0,Y 572.985,Z 277.734,A -85,B 0,C 180,E1 -2079.888,E2 -2079.888} C_VEL
LIN {X 0,Y 572.996,Z 274.2,A -85,B 0,C 180,E1 -2081.117,E2 -2081.117} C_VEL
LIN {X 0,Y 573.034,Z 269.04,A -85,B 0,C 180,E1 -2082.394,E2 -2082.394} C_VEL
LIN {X 0,Y 573.082,Z 263.339,A -85,B 0,C 180,E1 -2083.474,E2 -2083.474} C_VEL
LIN {X 0,Y 573.162,Z 256.194,A -85,B 0,C 180,E1 -2084.553,E2 -2084.553} C_VEL
LIN {X 0,Y 573.223,Z 247.102,A -85,B 0,C 180,E1 -2085.648,E2 -2085.648} C_VEL
LIN {X 0,Y 573.302,Z 237.967,A -85,B 0,C 180,E1 -2086.542,E2 -2086.542} C_VEL
LIN {X 0,Y 573.402,Z 227.315,A -85,B 0,C 180,E1 -2087.383,E2 -2087.383} C_VEL
LIN {X 0,Y 573.526,Z 215.622,A -85,B 0,C 180,E1 -2088.116,E2 -2088.116} C_VEL
LIN {X 0,Y 573.707,Z 203.36,A -85,B 0,C 180,E1 -2088.712,E2 -2088.712} C_VEL
LIN {X 0,Y 573.805,Z 190.319,A -85,B 0,C 180,E1 -2089.172,E2 -2089.172} C_VEL
LIN {X 0,Y 573.87,Z 177.388,A -85,B 0,C 180,E1 -2089.479,E2 -2089.479} C_VEL
LIN {X 0,Y 573.913,Z 74.495,A -85,B 0,C 180,E1 -2090.793,E2 -2090.793} C_VEL
LIN {X 0,Y 573.269,Z 70.607,A -85,B 0,C 180,E1 -2090.867,E2 -2090.867} C_VEL
LIN {X 0,Y 573.356,Z 55.644,A -85,B 0,C 180,E1 -2093.668,E2 -2093.668} C_VEL
LIN {X 0,Y 573.307,Z 46.478,A -85,B 0,C 180,E1 -2095.408,E2 -2095.408} C_VEL
LIN {X 0,Y 573.243,Z 46.08,A -85,B 0,C 180,E1 -2095.508,E2 -2095.508} C_VEL
LIN {X 0,Y 573.184,Z 46.089,A -85,B 0,C 180,E1 -2098.568,E2 -2098.568} C_VEL
LIN {X 0,Y 573.209,Z 46.08,A -85,B 0,C 180,E1 -2100.995,E2 -2100.995} C_VEL
LIN {X 0,Y 573.22,Z 46.079,A -85,B 0,C 180,E1 -2103.517,E2 -2103.517} C_VEL
LIN {X 0,Y 573.182,Z 46.091,A -85,B 0,C 180,E1 -2106.054,E2 -2106.054} C_VEL
LIN {X 0,Y 573.215,Z 46.079,A -85,B 0,C 180,E1 -2108.704,E2 -2108.704} C_VEL
LIN {X 0,Y 573.188,Z 46.086,A -85,B 0,C 180,E1 -2111.587,E2 -2111.587} C_VEL
LIN {X 0,Y 573.207,Z 46.079,A -85,B 0,C 180,E1 -2114.337,E2 -2114.337} C_VEL
LIN {X 0,Y 573.199,Z 46.08,A -85,B 0,C 180,E1 -2116.637,E2 -2116.637} C_VEL
LIN {X 0,Y 573.203,Z 46.086,A -85,B 0,C 180,E1 -2119.48,E2 -2119.48} C_VEL
LIN {X 0,Y 573.164,Z 46.085,A -85,B 0,C 180,E1 -2122.186,E2 -2122.186} C_VEL
LIN {X 0,Y 573.214,Z 46.084,A -85,B 0,C 180,E1 -2125.232,E2 -2125.232} C_VEL
LIN {X 0,Y 573.22,Z 46.076,A -85,B 0,C 180,E1 -2128.183,E2 -2128.183} C_VEL
LIN {X 0,Y 573.228,Z 46.078,A -85,B 0,C 180,E1 -2130.632,E2 -2130.632} C_VEL
LIN {X 0,Y 573.195,Z 46.084,A -85,B 0,C 180,E1 -2133.517,E2 -2133.517} C_VEL
LIN {X 0,Y 573.193,Z 46.08,A -85,B 0,C 180,E1 -2136.133,E2 -2136.133} C_VEL
LIN {X 0,Y 573.246,Z 46.079,A -85,B 0,C 180,E1 -2139.173,E2 -2139.173} C_VEL
LIN {X 0,Y 573.203,Z 46.08,A -85,B 0,C 180,E1 -2141.41,E2 -2141.41} C_VEL
LIN {X 0,Y 573.226,Z 46.076,A -85,B 0,C 180,E1 -2143.621,E2 -2143.621} C_VEL
LIN {X 0,Y 573.2,Z 46.087,A -85,B 0,C 180,E1 -2146.528,E2 -2146.528} C_VEL
LIN {X 0,Y 573.239,Z 46.074,A -85,B 0,C 180,E1 -2149.403,E2 -2149.403} C_VEL
LIN {X 0,Y 573.239,Z 46.081,A -85,B 0,C 180,E1 -2152.249,E2 -2152.249} C_VEL
LIN {X 0,Y 573.284,Z 46.069,A -85,B 0,C 180,E1 -2155.077,E2 -2155.077} C_VEL
LIN {X 0,Y 573.297,Z 46.071,A -85,B 0,C 180,E1 -2157.892,E2 -2157.892} C_VEL
LIN {X 0,Y 573.327,Z 46.065,A -85,B 0,C 180,E1 -2160.702,E2 -2160.702} C_VEL
LIN {X 0,Y 573.29,Z 46.069,A -85,B 0,C 180,E1 -2162.811,E2 -2162.811} C_VEL
LIN {X 0,Y 573.272,Z 46.074,A -85,B 0,C 180,E1 -2165.628,E2 -2165.628} C_VEL
LIN {X 0,Y 573.251,Z 46.075,A -85,B 0,C 180,E1 -2168.46,E2 -2168.46} C_VEL
LIN {X 0,Y 573.276,Z 46.072,A -85,B 0,C 180,E1 -2171.312,E2 -2171.312} C_VEL
LIN {X 0,Y 573.274,Z 46.071,A -85,B 0,C 180,E1 -2174.42,E2 -2174.42} C_VEL
LIN {X 0,Y 573.241,Z 46.076,A -85,B 0,C 180,E1 -2177.112,E2 -2177.112} C_VEL
LIN {X 0,Y 573.237,Z 46.076,A -85,B 0,C 180,E1 -2180.077,E2 -2180.077} C_VEL
LIN {X 0,Y 573.224,Z 46.075,A -85,B 0,C 180,E1 -2182.338,E2 -2182.338} C_VEL
LIN {X 0,Y 573.238,Z 46.082,A -85,B 0,C 180,E1 -2185.411,E2 -2185.411} C_VEL
LIN {X 0,Y 573.232,Z 46.077,A -85,B 0,C 180,E1 -2188.565,E2 -2188.565} C_VEL
LIN {X 0,Y 573.221,Z 46.085,A -85,B 0,C 180,E1 -2190.994,E2 -2190.994} C_VEL
LIN {X 0,Y 573.266,Z 46.073,A -85,B 0,C 180,E1 -2193.524,E2 -2193.524} C_VEL
LIN {X 0,Y 573.217,Z 46.075,A -85,B 0,C 180,E1 -2196.051,E2 -2196.051} C_VEL
LIN {X 0,Y 573.24,Z 46.082,A -85,B 0,C 180,E1 -2198.702,E2 -2198.702} C_VEL
LIN {X 0,Y 573.23,Z 46.076,A -85,B 0,C 180,E1 -2201.592,E2 -2201.592} C_VEL
LIN {X 0,Y 573.225,Z 46.082,A -85,B 0,C 180,E1 -2204.335,E2 -2204.335} C_VEL
LIN {X 0,Y 573.242,Z 46.074,A -85,B 0,C 180,E1 -2207.359,E2 -2207.359} C_VEL
LIN {X 0,Y 573.248,Z 46.082,A -85,B 0,C 180,E1 -2210.393,E2 -2210.393} C_VEL
LIN {X 0,Y 573.255,Z 46.073,A -85,B 0,C 180,E1 -2213.077,E2 -2213.077} C_VEL
LIN {X 0,Y 573.269,Z 46.073,A -85,B 0,C 180,E1 -2215.671,E2 -2215.671} C_VEL
LIN {X 0,Y 573.242,Z 46.084,A -85,B 0,C 180,E1 -2218.184,E2 -2218.184} C_VEL
LIN {X 0,Y 573.264,Z 46.074,A -85,B 0,C 180,E1 -2220.634,E2 -2220.634} C_VEL
LIN {X 0,Y 573.253,Z 46.074,A -85,B 0,C 180,E1 -2223.024,E2 -2223.024} C_VEL
LIN {X 0,Y 573.279,Z 46.074,A -85,B 0,C 180,E1 -2225.366,E2 -2225.366} C_VEL
LIN {X 0,Y 573.282,Z 46.202,A -85,B 0,C 180,E1 -2226.204,E2 -2226.204} C_VEL
LIN {X 0,Y 573.943,Z 51.18,A -85,B 0,C 180,E1 -2226.93,E2 -2226.93} C_VEL
LIN {X 0,Y 573.784,Z 68.804,A -85,B 0,C 180,E1 -2229.381,E2 -2229.381} C_VEL
LIN {X 0,Y 573.638,Z 89.13,A -85,B 0,C 180,E1 -2232.164,E2 -2232.164} C_VEL
LIN {X 0,Y 573.458,Z 107.966,A -85,B 0,C 180,E1 -2234.722,E2 -2234.722} C_VEL
LIN {X 0,Y 573.4,Z 118.52,A -85,B 0,C 180,E1 -2236.161,E2 -2236.161} C_VEL
LIN {X 0,Y 574.058,Z 124.489,A -85,B 0,C 180,E1 -2236.256,E2 -2236.256} C_VEL
LIN {X 0,Y 573.894,Z 226.934,A -85,B 0,C 180,E1 -2237.557,E2 -2237.557} C_VEL
LIN {X 0,Y 573.807,Z 240.209,A -85,B 0,C 180,E1 -2237.87,E2 -2237.87} C_VEL
LIN {X 0,Y 573.7,Z 252.372,A -85,B 0,C 180,E1 -2238.294,E2 -2238.294} C_VEL
LIN {X 0,Y 573.567,Z 264.62,A -85,B 0,C 180,E1 -2238.873,E2 -2238.873} C_VEL
LIN {X 0,Y 573.426,Z 276.193,A -85,B 0,C 180,E1 -2239.585,E2 -2239.585} C_VEL
LIN {X 0,Y 573.333,Z 286.601,A -85,B 0,C 180,E1 -2240.385,E2 -2240.385} C_VEL
LIN {X 0,Y 573.241,Z 295.111,A -85,B 0,C 180,E1 -2241.184,E2 -2241.184} C_VEL
LIN {X 0,Y 573.161,Z 302.959,A -85,B 0,C 180,E1 -2242.071,E2 -2242.071} C_VEL
LIN {X 0,Y 573.073,Z 310.58,A -85,B 0,C 180,E1 -2243.126,E2 -2243.126} C_VEL
LIN {X 0,Y 573.07,Z 317.679,A -85,B 0,C 180,E1 -2244.369,E2 -2244.369} C_VEL
LIN {X 0,Y 573.028,Z 322.372,A -85,B 0,C 180,E1 -2245.427,E2 -2245.427} C_VEL
LIN {X 0,Y 573.022,Z 325.957,A -85,B 0,C 180,E1 -2246.484,E2 -2246.484} C_VEL
LIN {X 0,Y 572.959,Z 327.807,A -85,B 0,C 180,E1 -2247.187,E2 -2247.187} C_VEL
LIN {X 0,Y 572.946,Z 330.184,A -85,B 0,C 180,E1 -2248.594,E2 -2248.594} C_VEL
LIN {X 0,Y 572.938,Z 331,A -85,B 0,C 180,E1 -2250,E2 -2250} C_VEL
LIN {X 0,Y 572.946,Z 330.186,A -85,B 0,C 180,E1 -2251.406,E2 -2251.406} C_VEL
LIN {X 0,Y 572.959,Z 327.81,A -85,B 0,C 180,E1 -2252.812,E2 -2252.812} C_VEL
LIN {X 0,Y 573.014,Z 324.896,A -85,B 0,C 180,E1 -2253.868,E2 -2253.868} C_VEL
LIN {X 0,Y 572.963,Z 320.949,A -85,B 0,C 180,E1 -2254.925,E2 -2254.925} C_VEL
LIN {X 0,Y 573.093,Z 315.868,A -85,B 0,C 180,E1 -2255.983,E2 -2255.983} C_VEL
LIN {X 0,Y 573.103,Z 309.469,A -85,B 0,C 180,E1 -2257.044,E2 -2257.044} C_VEL
LIN {X 0,Y 573.177,Z 301.479,A -85,B 0,C 180,E1 -2258.106,E2 -2258.106} C_VEL
LIN {X 0,Y 573.254,Z 293.336,A -85,B 0,C 180,E1 -2258.993,E2 -2258.993} C_VEL
LIN {X 0,Y 573.346,Z 283.401,A -85,B 0,C 180,E1 -2259.881,E2 -2259.881} C_VEL
LIN {X 0,Y 573.501,Z 272.214,A -85,B 0,C 180,E1 -2260.679,E2 -2260.679} C_VEL
LIN {X 0,Y 573.586,Z 261.177,A -85,B 0,C 180,E1 -2261.306,E2 -2261.306} C_VEL
LIN {X 0,Y 573.7,Z 248.984,A -85,B 0,C 180,E1 -2261.84,E2 -2261.84} C_VEL
LIN {X 0,Y 573.828,Z 236.182,A -85,B 0,C 180,E1 -2262.241,E2 -2262.241} C_VEL
LIN {X 0,Y 573.88,Z 222.613,A -85,B 0,C 180,E1 -2262.51,E2 -2262.51} C_VEL
